LIN {X 0,Y 320.204,Z 957.496,A -85,B 0,C 180,E1 15355.155,E2 15355.155} C_VEL
LIN {X 0,Y 325.919,Z 943.483,A -85,B 0,C 180,E1 15351.712,E2 15351.712} C_VEL
LIN {X 0,Y 332.277,Z 928.194,A -85,B 0,C 180,E1 15348.526,E2 15348.526} C_VEL
LIN {X 0,Y 338.79,Z 912.192,A -85,B 0,C 180,E1 15345.742,E2 15345.742} C_VEL
LIN {X 0,Y 346.075,Z 893.682,A -85,B 0,C 180,E1 15343.041,E2 15343.041} C_VEL
LIN {X 0,Y 352.439,Z 876.534,A -85,B 0,C 180,E1 15340.945,E2 15340.945} C_VEL
LIN {X 0,Y 359.474,Z 856.024,A -85,B 0,C 180,E1 15338.858,E2 15338.858} C_VEL
LIN {X 0,Y 365.817,Z 835.8,A -85,B 0,C 180,E1 15337.159,E2 15337.159} C_VEL
LIN {X 0,Y 371.591,Z 814.628,A -85,B 0,C 180,E1 15335.724,E2 15335.724} C_VEL
LIN {X 0,Y 376.805,Z 792.847,A -85,B 0,C 180,E1 15334.531,E2 15334.531} C_VEL
LIN {X 0,Y 381.083,Z 770.761,A -85,B 0,C 180,E1 15333.6,E2 15333.6} C_VEL
LIN {X 0,Y 384.81,Z 746.357,A -85,B 0,C 180,E1 15332.838,E2 15332.838} C_VEL
LIN {X 0,Y 387.003,Z 723.943,A -85,B 0,C 180,E1 15332.314,E2 15332.314} C_VEL
LIN {X 0,Y 400.127,Z 517.073,A -85,B 0,C 180,E1 15328.257,E2 15328.257} C_VEL
LIN {X 0,Y 400.762,Z 506.979,A -85,B 0,C 180,E1 15328.052,E2 15328.052} C_VEL
LIN {X 0,Y 392.665,Z 493.102,A -85,B 0,C 180,E1 15325.206,E2 15325.206} C_VEL
LIN {X 0,Y 385.414,Z 481.504,A -85,B 0,C 180,E1 15322.297,E2 15322.297} C_VEL
LIN {X 0,Y 380.756,Z 474.893,A -85,B 0,C 180,E1 15320.201,E2 15320.201} C_VEL
LIN {X 0,Y 377.273,Z 470.183,A -85,B 0,C 180,E1 15318.463,E2 15318.463} C_VEL
LIN {X 0,Y 373.457,Z 465.169,A -85,B 0,C 180,E1 15316.326,E2 15316.326} C_VEL
LIN {X 0,Y 370.115,Z 460.624,A -85,B 0,C 180,E1 15314.151,E2 15314.151} C_VEL
LIN {X 0,Y 366.362,Z 456.303,A -85,B 0,C 180,E1 15311.252,E2 15311.252} C_VEL
LIN {X 0,Y 365.344,Z 454.428,A -85,B 0,C 180,E1 15310.246,E2 15310.246} C_VEL
LIN {X 0,Y 362.011,Z 451.144,A -85,B 0,C 180,E1 15306.342,E2 15306.342} C_VEL
LIN {X 0,Y 360.93,Z 448.352,A -85,B 0,C 180,E1 15303.971,E2 15303.971} C_VEL
LIN {X 0,Y 360.463,Z 448.211,A -85,B 0,C 180,E1 15296.66,E2 15296.66} C_VEL
LIN {X 0,Y 361.126,Z 448.613,A -85,B 0,C 180,E1 15294.996,E2 15294.996} C_VEL
LIN {X 0,Y 362.687,Z 452.129,A -85,B 0,C 180,E1 15292.077,E2 15292.077} C_VEL
LIN {X 0,Y 365.646,Z 454.865,A -85,B 0,C 180,E1 15288.884,E2 15288.884} C_VEL
LIN {X 0,Y 368.285,Z 458.822,A -85,B 0,C 180,E1 15286.578,E2 15286.578} C_VEL
LIN {X 0,Y 370.2,Z 460.795,A -85,B 0,C 180,E1 15285.212,E2 15285.212} C_VEL
LIN {X 0,Y 373.571,Z 465.247,A -85,B 0,C 180,E1 15283.038,E2 15283.038} C_VEL
LIN {X 0,Y 378.886,Z 472.366,A -85,B 0,C 180,E1 15280.137,E2 15280.137} C_VEL
LIN {X 0,Y 382.899,Z 477.884,A -85,B 0,C 180,E1 15278.235,E2 15278.235} C_VEL
LIN {X 0,Y 388.744,Z 485.936,A -85,B 0,C 180,E1 15275.78,E2 15275.78} C_VEL
LIN {X 0,Y 397.542,Z 499.019,A -85,B 0,C 180,E1 15272.555,E2 15272.555} C_VEL
LIN {X 0,Y 400.68,Z 504.305,A -85,B 0,C 180,E1 15271.496,E2 15271.496} C_VEL
LIN {X 0,Y 387.414,Z 710.788,A -85,B 0,C 180,E1 15267.448,E2 15267.448} C_VEL
LIN {X 0,Y 385.19,Z 733.04,A -85,B 0,C 180,E1 15266.904,E2 15266.904} C_VEL
LIN {X 0,Y 381.856,Z 755.375,A -85,B 0,C 180,E1 15266.142,E2 15266.142} C_VEL
LIN {X 0,Y 377.948,Z 776.257,A -85,B 0,C 180,E1 15265.218,E2 15265.218} C_VEL
LIN {X 0,Y 373.062,Z 797.329,A -85,B 0,C 180,E1 15264.028,E2 15264.028} C_VEL
LIN {X 0,Y 367.712,Z 817.41,A -85,B 0,C 180,E1 15262.642,E2 15262.642} C_VEL
LIN {X 0,Y 361.615,Z 837.121,A -85,B 0,C 180,E1 15260.974,E2 15260.974} C_VEL
LIN {X 0,Y 355.259,Z 855.944,A -85,B 0,C 180,E1 15259.074,E2 15259.074} C_VEL
LIN {X 0,Y 348.293,Z 874.444,A -85,B 0,C 180,E1 15256.809,E2 15256.809} C_VEL
LIN {X 0,Y 341.213,Z 892.21,A -85,B 0,C 180,E1 15254.213,E2 15254.213} C_VEL
LIN {X 0,Y 334.762,Z 907.539,A -85,B 0,C 180,E1 15251.527,E2 15251.527} C_VEL
LIN {X 0,Y 327.933,Z 923.307,A -85,B 0,C 180,E1 15248.233,E2 15248.233} C_VEL
LIN {X 0,Y 322.331,Z 936.215,A -85,B 0,C 180,E1 15245.015,E2 15245.015} C_VEL
LIN {X 0,Y 316.952,Z 948.748,A -85,B 0,C 180,E1 15241.251,E2 15241.251} C_VEL
LIN {X 0,Y 312.67,Z 959.438,A -85,B 0,C 180,E1 15237.414,E2 15237.414} C_VEL
LIN {X 0,Y 309.22,Z 968.65,A -85,B 0,C 180,E1 15233.319,E2 15233.319} C_VEL
LIN {X 0,Y 306.721,Z 976.512,A -85,B 0,C 180,E1 15229.022,E2 15229.022} C_VEL
LIN {X 0,Y 305.297,Z 981.991,A -85,B 0,C 180,E1 15225.187,E2 15225.187} C_VEL
LIN {X 0,Y 304.432,Z 986.613,A -85,B 0,C 180,E1 15220.98,E2 15220.98} C_VEL
LIN {X 0,Y 304.083,Z 989.403,A -85,B 0,C 180,E1 15217.176,E2 15217.176} C_VEL
LIN {X 0,Y 303.978,Z 991.015,A -85,B 0,C 180,E1 15213.582,E2 15213.582} C_VEL
LIN {X 0,Y 303.96,Z 991.586,A -85,B 0,C 180,E1 15209.623,E2 15209.623} C_VEL
LIN {X 0,Y 303.993,Z 990.851,A -85,B 0,C 180,E1 15205.85,E2 15205.85} C_VEL
LIN {X 0,Y 304.109,Z 989.131,A -85,B 0,C 180,E1 15202.253,E2 15202.253} C_VEL
LIN {X 0,Y 304.564,Z 985.749,A -85,B 0,C 180,E1 15198.045,E2 15198.045} C_VEL
LIN {X 0,Y 305.44,Z 981.375,A -85,B 0,C 180,E1 15194.236,E2 15194.236} C_VEL
LIN {X 0,Y 305.492,Z 981.166,A -85,B 0,C 180,E1 15194.073,E2 15194.073} C_VEL
LIN {X 0,Y 305.002,Z 979.368,A -85,B 0,C 180,E1 15192.66,E2 15192.66} C_VEL
LIN {X 0,Y 300.55,Z 974.185,A -85,B 0,C 180,E1 15188.845,E2 15188.845} C_VEL
LIN {X 0,Y 300.527,Z 972.173,A -85,B 0,C 180,E1 15187.629,E2 15187.629} C_VEL
LIN {X 0,Y 303.768,Z 963.538,A -85,B 0,C 180,E1 15183.41,E2 15183.41} C_VEL
LIN {X 0,Y 307.801,Z 953.96,A -85,B 0,C 180,E1 15179.556,E2 15179.556} C_VEL
LIN {X 0,Y 312.845,Z 942.539,A -85,B 0,C 180,E1 15175.775,E2 15175.775} C_VEL
LIN {X 0,Y 318.733,Z 929.796,A -85,B 0,C 180,E1 15172.234,E2 15172.234} C_VEL
LIN {X 0,Y 325.37,Z 915.155,A -85,B 0,C 180,E1 15168.887,E2 15168.887} C_VEL
LIN {X 0,Y 332.637,Z 898.955,A -85,B 0,C 180,E1 15165.79,E2 15165.79} C_VEL
LIN {X 0,Y 339.295,Z 883.331,A -85,B 0,C 180,E1 15163.298,E2 15163.298} C_VEL
LIN {X 0,Y 346.999,Z 864.093,A -85,B 0,C 180,E1 15160.735,E2 15160.735} C_VEL
LIN {X 0,Y 353.709,Z 845.967,A -85,B 0,C 180,E1 15158.729,E2 15158.729} C_VEL
LIN {X 0,Y 360.218,Z 826.344,A -85,B 0,C 180,E1 15156.935,E2 15156.935} C_VEL
LIN {X 0,Y 366.181,Z 806.306,A -85,B 0,C 180,E1 15155.416,E2 15155.416} C_VEL
LIN {X 0,Y 371.435,Z 785.463,A -85,B 0,C 180,E1 15154.14,E2 15154.14} C_VEL
LIN {X 0,Y 376.179,Z 763.349,A -85,B 0,C 180,E1 15153.053,E2 15153.053} C_VEL
LIN {X 0,Y 379.818,Z 741.232,A -85,B 0,C 180,E1 15152.229,E2 15152.229} C_VEL
LIN {X 0,Y 382.735,Z 717.296,A -85,B 0,C 180,E1 15151.579,E2 15151.579} C_VEL
LIN {X 0,Y 395.368,Z 528.784,A -85,B 0,C 180,E1 15147.863,E2 15147.863} C_VEL
LIN {X 0,Y 396.731,Z 508.619,A -85,B 0,C 180,E1 15147.465,E2 15147.465} C_VEL
LIN {X 0,Y 389.098,Z 496.82,A -85,B 0,C 180,E1 15144.682,E2 15144.682} C_VEL
LIN {X 0,Y 382.445,Z 487.221,A -85,B 0,C 180,E1 15141.914,E2 15141.914} C_VEL
LIN {X 0,Y 378.4,Z 481.609,A -85,B 0,C 180,E1 15140.01,E2 15140.01} C_VEL
LIN {X 0,Y 375.455,Z 477.526,A -85,B 0,C 180,E1 15138.476,E2 15138.476} C_VEL
LIN {X 0,Y 372.006,Z 472.824,A -85,B 0,C 180,E1 15136.473,E2 15136.473} C_VEL
LIN {X 0,Y 368.649,Z 468.169,A -85,B 0,C 180,E1 15134.209,E2 15134.209} C_VEL
LIN {X 0,Y 365.046,Z 463.88,A -85,B 0,C 180,E1 15131.294,E2 15131.294} C_VEL
LIN {X 0,Y 364.061,Z 462.185,A -85,B 0,C 180,E1 15130.284,E2 15130.284} C_VEL
LIN {X 0,Y 360.943,Z 458.912,A -85,B 0,C 180,E1 15126.362,E2 15126.362} C_VEL
LIN {X 0,Y 360.04,Z 456.293,A -85,B 0,C 180,E1 15124.141,E2 15124.141} C_VEL
LIN {X 0,Y 359.977,Z 456.281,A -85,B 0,C 180,E1 15116.497,E2 15116.497} C_VEL
LIN {X 0,Y 362.455,Z 460.975,A -85,B 0,C 180,E1 15111.913,E2 15111.913} C_VEL
LIN {X 0,Y 364.452,Z 462.647,A -85,B 0,C 180,E1 15109.808,E2 15109.808} C_VEL
LIN {X 0,Y 367.084,Z 466.751,A -85,B 0,C 180,E1 15107.415,E2 15107.415} C_VEL
LIN {X 0,Y 368.85,Z 468.542,A -85,B 0,C 180,E1 15106.12,E2 15106.12} C_VEL
LIN {X 0,Y 372.256,Z 473.092,A -85,B 0,C 180,E1 15103.86,E2 15103.86} C_VEL
LIN {X 0,Y 377.256,Z 479.962,A -85,B 0,C 180,E1 15101.055,E2 15101.055} C_VEL
LIN {X 0,Y 381.18,Z 485.5,A -85,B 0,C 180,E1 15099.141,E2 15099.141} C_VEL
LIN {X 0,Y 385.654,Z 492.449,A -85,B 0,C 180,E1 15097.155,E2 15097.155} C_VEL
LIN {X 0,Y 392.548,Z 503.898,A -85,B 0,C 180,E1 15094.423,E2 15094.423} C_VEL
LIN {X 0,Y 396.813,Z 511.775,A -85,B 0,C 180,E1 15092.873,E2 15092.873} C_VEL
LIN {X 0,Y 383.039,Z 721.232,A -85,B 0,C 180,E1 15088.764,E2 15088.764} C_VEL
LIN {X 0,Y 380.765,Z 744.543,A -85,B 0,C 180,E1 15088.226,E2 15088.226} C_VEL
LIN {X 0,Y 377.031,Z 768.994,A -85,B 0,C 180,E1 15087.482,E2 15087.482} C_VEL
LIN {X 0,Y 373.092,Z 788.994,A -85,B 0,C 180,E1 15086.662,E2 15086.662} C_VEL
LIN {X 0,Y 367.684,Z 811.66,A -85,B 0,C 180,E1 15085.474,E2 15085.474} C_VEL
LIN {X 0,Y 362.223,Z 831.325,A -85,B 0,C 180,E1 15084.184,E2 15084.184} C_VEL
LIN {X 0,Y 355.5,Z 852.565,A -85,B 0,C 180,E1 15082.472,E2 15082.472} C_VEL
LIN {X 0,Y 348.764,Z 871.867,A -85,B 0,C 180,E1 15080.582,E2 15080.582} C_VEL
LIN {X 0,Y 341.43,Z 890.989,A -85,B 0,C 180,E1 15078.303,E2 15078.303} C_VEL
LIN {X 0,Y 334.217,Z 908.855,A -85,B 0,C 180,E1 15075.76,E2 15075.76} C_VEL
LIN {X 0,Y 327.211,Z 925.222,A -85,B 0,C 180,E1 15072.949,E2 15072.949} C_VEL
LIN {X 0,Y 320.072,Z 941.638,A -85,B 0,C 180,E1 15069.583,E2 15069.583} C_VEL
LIN {X 0,Y 314.248,Z 955.086,A -85,B 0,C 180,E1 15066.281,E2 15066.281} C_VEL
LIN {X 0,Y 308.813,Z 967.94,A -85,B 0,C 180,E1 15062.508,E2 15062.508} C_VEL
LIN {X 0,Y 304.281,Z 979.499,A -85,B 0,C 180,E1 15058.452,E2 15058.452} C_VEL
LIN {X 0,Y 300.872,Z 989.048,A -85,B 0,C 180,E1 15054.333,E2 15054.333} C_VEL
LIN {X 0,Y 298.43,Z 997.374,A -85,B 0,C 180,E1 15049.981,E2 15049.981} C_VEL
LIN {X 0,Y 296.983,Z 1003.564,A -85,B 0,C 180,E1 15045.824,E2 15045.824} C_VEL
LIN {X 0,Y 296.221,Z 1008.587,A -85,B 0,C 180,E1 15041.486,E2 15041.486} C_VEL
LIN {X 0,Y 295.976,Z 1011.635,A -85,B 0,C 180,E1 15037.57,E2 15037.57} C_VEL
LIN {X 0,Y 295.96,Z 1013.344,A -85,B 0,C 180,E1 15034.068,E2 15034.068} C_VEL
LIN {X 0,Y 295.977,Z 1014.117,A -85,B 0,C 180,E1 15030.001,E2 15030.001} C_VEL
LIN {X 0,Y 295.959,Z 1013.342,A -85,B 0,C 180,E1 15025.933,E2 15025.933} C_VEL
LIN {X 0,Y 295.977,Z 1011.631,A -85,B 0,C 180,E1 15022.431,E2 15022.431} C_VEL
LIN {X 0,Y 296.241,Z 1008.39,A -85,B 0,C 180,E1 15018.318,E2 15018.318} C_VEL
LIN {X 0,Y 296.982,Z 1003.558,A -85,B 0,C 180,E1 15014.177,E2 15014.177} C_VEL
LIN {X 0,Y 298.428,Z 997.364,A -85,B 0,C 180,E1 15010.02,E2 15010.02} C_VEL
LIN {X 0,Y 300.874,Z 989.034,A -85,B 0,C 180,E1 15005.668,E2 15005.668} C_VEL
LIN {X 0,Y 304.278,Z 979.484,A -85,B 0,C 180,E1 15001.549,E2 15001.549} C_VEL
LIN {X 0,Y 308.808,Z 967.92,A -85,B 0,C 180,E1 14997.493,E2 14997.493} C_VEL
LIN {X 0,Y 314.542,Z 954.339,A -85,B 0,C 180,E1 14993.533,E2 14993.533} C_VEL
LIN {X 0,Y 320.416,Z 940.813,A -85,B 0,C 180,E1 14990.237,E2 14990.237} C_VEL
LIN {X 0,Y 327.404,Z 924.699,A -85,B 0,C 180,E1 14986.964,E2 14986.964} C_VEL
LIN {X 0,Y 334.431,Z 908.269,A -85,B 0,C 180,E1 14984.155,E2 14984.155} C_VEL
LIN {X 0,Y 341.586,Z 890.474,A -85,B 0,C 180,E1 14981.64,E2 14981.64} C_VEL
LIN {X 0,Y 349.009,Z 871.012,A -85,B 0,C 180,E1 14979.339,E2 14979.339} C_VEL
LIN {X 0,Y 355.484,Z 852.438,A -85,B 0,C 180,E1 14977.526,E2 14977.526} C_VEL
LIN {X 0,Y 362.323,Z 830.765,A -85,B 0,C 180,E1 14975.785,E2 14975.785} C_VEL
LIN {X 0,Y 367.666,Z 811.477,A -85,B 0,C 180,E1 14974.523,E2 14974.523} C_VEL
LIN {X 0,Y 372.9,Z 789.56,A -85,B 0,C 180,E1 14973.371,E2 14973.371} C_VEL
LIN {X 0,Y 376.938,Z 769.089,A -85,B 0,C 180,E1 14972.529,E2 14972.529} C_VEL
LIN {X 0,Y 380.682,Z 744.574,A -85,B 0,C 180,E1 14971.782,E2 14971.782} C_VEL
LIN {X 0,Y 382.974,Z 721.037,A -85,B 0,C 180,E1 14971.24,E2 14971.24} C_VEL
LIN {X 0,Y 396.738,Z 511.466,A -85,B 0,C 180,E1 14967.129,E2 14967.129} C_VEL
LIN {X 0,Y 389.576,Z 498.912,A -85,B 0,C 180,E1 14964.487,E2 14964.487} C_VEL
LIN {X 0,Y 382.313,Z 487.129,A -85,B 0,C 180,E1 14961.433,E2 14961.433} C_VEL
LIN {X 0,Y 378.126,Z 481.293,A -85,B 0,C 180,E1 14959.461,E2 14959.461} C_VEL
LIN {X 0,Y 375.458,Z 477.57,A -85,B 0,C 180,E1 14958.074,E2 14958.074} C_VEL
LIN {X 0,Y 371.857,Z 472.733,A -85,B 0,C 180,E1 14955.998,E2 14955.998} C_VEL
LIN {X 0,Y 368.172,Z 467.718,A -85,B 0,C 180,E1 14953.506,E2 14953.506} C_VEL
LIN {X 0,Y 365.12,Z 464.139,A -85,B 0,C 180,E1 14951.051,E2 14951.051} C_VEL
LIN {X 0,Y 364.041,Z 462.222,A -85,B 0,C 180,E1 14949.964,E2 14949.964} C_VEL
LIN {X 0,Y 360.758,Z 458.669,A -85,B 0,C 180,E1 14945.885,E2 14945.885} C_VEL
LIN {X 0,Y 359.886,Z 456.277,A -85,B 0,C 180,E1 14943.823,E2 14943.823} C_VEL
LIN {X 0,Y 359.49,Z 456.153,A -85,B 0,C 180,E1 14936.651,E2 14936.651} C_VEL
LIN {X 0,Y 360.073,Z 456.551,A -85,B 0,C 180,E1 14935.141,E2 14935.141} C_VEL
LIN {X 0,Y 361.71,Z 460.167,A -85,B 0,C 180,E1 14932.055,E2 14932.055} C_VEL
LIN {X 0,Y 364.345,Z 462.578,A -85,B 0,C 180,E1 14929.165,E2 14929.165} C_VEL
LIN {X 0,Y 367.015,Z 466.623,A -85,B 0,C 180,E1 14926.771,E2 14926.771} C_VEL
LIN {X 0,Y 368.784,Z 468.533,A -85,B 0,C 180,E1 14925.476,E2 14925.476} C_VEL
LIN {X 0,Y 372.353,Z 473.176,A -85,B 0,C 180,E1 14923.141,E2 14923.141} C_VEL
LIN {X 0,Y 377.32,Z 480.16,A -85,B 0,C 180,E1 14920.374,E2 14920.374} C_VEL
LIN {X 0,Y 381.277,Z 485.71,A -85,B 0,C 180,E1 14918.461,E2 14918.461} C_VEL
LIN {X 0,Y 386.702,Z 493.369,A -85,B 0,C 180,E1 14916.131,E2 14916.131} C_VEL
LIN {X 0,Y 394.978,Z 505.909,A -85,B 0,C 180,E1 14913.015,E2 14913.015} C_VEL
LIN {X 0,Y 396.636,Z 508.825,A -85,B 0,C 180,E1 14912.429,E2 14912.429} C_VEL
LIN {X 0,Y 382.999,Z 713.139,A -85,B 0,C 180,E1 14908.413,E2 14908.413} C_VEL
LIN {X 0,Y 380.495,Z 736.296,A -85,B 0,C 180,E1 14907.828,E2 14907.828} C_VEL
LIN {X 0,Y 377.14,Z 757.433,A -85,B 0,C 180,E1 14907.084,E2 14907.084} C_VEL
LIN {X 0,Y 372.84,Z 779.225,A -85,B 0,C 180,E1 14906.096,E2 14906.096} C_VEL
LIN {X 0,Y 368.092,Z 798.762,A -85,B 0,C 180,E1 14904.972,E2 14904.972} C_VEL
LIN {X 0,Y 362.377,Z 819.346,A -85,B 0,C 180,E1 14903.533,E2 14903.533} C_VEL
LIN {X 0,Y 356.288,Z 838.235,A -85,B 0,C 180,E1 14901.913,E2 14901.913} C_VEL
LIN {X 0,Y 349.442,Z 857.624,A -85,B 0,C 180,E1 14899.925,E2 14899.925} C_VEL
LIN {X 0,Y 342.507,Z 875.356,A -85,B 0,C 180,E1 14897.726,E2 14897.726} C_VEL
LIN {X 0,Y 334.93,Z 893.521,A -85,B 0,C 180,E1 14895.025,E2 14895.025} C_VEL
LIN {X 0,Y 328.24,Z 908.763,A -85,B 0,C 180,E1 14892.307,E2 14892.307} C_VEL
LIN {X 0,Y 321.133,Z 924.376,A -85,B 0,C 180,E1 14888.966,E2 14888.966} C_VEL
LIN {X 0,Y 314.996,Z 937.894,A -85,B 0,C 180,E1 14885.507,E2 14885.507} C_VEL
LIN {X 0,Y 309.541,Z 949.889,A -85,B 0,C 180,E1 14881.765,E2 14881.765} C_VEL
LIN {X 0,Y 304.921,Z 960.735,A -85,B 0,C 180,E1 14877.705,E2 14877.705} C_VEL
LIN {X 0,Y 301.465,Z 969.527,A -85,B 0,C 180,E1 14873.657,E2 14873.657} C_VEL
LIN {X 0,Y 298.79,Z 977.408,A -85,B 0,C 180,E1 14869.141,E2 14869.141} C_VEL
LIN {X 0,Y 297.313,Z 982.841,A -85,B 0,C 180,E1 14865.164,E2 14865.164} C_VEL
LIN {X 0,Y 296.401,Z 987.378,A -85,B 0,C 180,E1 14860.69,E2 14860.69} C_VEL
LIN {X 0,Y 296.088,Z 989.923,A -85,B 0,C 180,E1 14856.981,E2 14856.981} C_VEL
LIN {X 0,Y 295.978,Z 991.578,A -85,B 0,C 180,E1 14852.904,E2 14852.904} C_VEL
LIN {X 0,Y 295.97,Z 991.797,A -85,B 0,C 180,E1 14848.838,E2 14848.838} C_VEL
LIN {X 0,Y 296.012,Z 990.956,A -85,B 0,C 180,E1 14845.156,E2 14845.156} C_VEL
LIN {X 0,Y 296.246,Z 988.685,A -85,B 0,C 180,E1 14840.873,E2 14840.873} C_VEL
LIN {X 0,Y 296.826,Z 985.074,A -85,B 0,C 180,E1 14836.759,E2 14836.759} C_VEL
LIN {X 0,Y 298.103,Z 979.901,A -85,B 0,C 180,E1 14832.432,E2 14832.432} C_VEL
LIN {X 0,Y 300.117,Z 973.342,A -85,B 0,C 180,E1 14828.299,E2 14828.299} C_VEL
LIN {X 0,Y 300.527,Z 972.173,A -85,B 0,C 180,E1 14827.629,E2 14827.629} C_VEL
LIN {X 0,Y 300.487,Z 969.761,A -85,B 0,C 180,E1 14826.222,E2 14826.222} C_VEL
LIN {X 0,Y 297.448,Z 963.001,A -85,B 0,C 180,E1 14822.402,E2 14822.402} C_VEL
LIN {X 0,Y 297.9,Z 960.498,A -85,B 0,C 180,E1 14821.214,E2 14821.214} C_VEL
LIN {X 0,Y 302.703,Z 949.892,A -85,B 0,C 180,E1 14817.204,E2 14817.204} C_VEL
LIN {X 0,Y 308.491,Z 937.836,A -85,B 0,C 180,E1 14813.394,E2 14813.394} C_VEL
LIN {X 0,Y 314.996,Z 924.269,A -85,B 0,C 180,E1 14809.887,E2 14809.887} C_VEL
LIN {X 0,Y 322.462,Z 908.563,A -85,B 0,C 180,E1 14806.506,E2 14806.506} C_VEL
LIN {X 0,Y 329.485,Z 893.265,A -85,B 0,C 180,E1 14803.767,E2 14803.767} C_VEL
LIN {X 0,Y 337.154,Z 875.582,A -85,B 0,C 180,E1 14801.133,E2 14801.133} C_VEL
LIN {X 0,Y 344.109,Z 858.451,A -85,B 0,C 180,E1 14798.997,E2 14798.997} C_VEL
LIN {X 0,Y 351.174,Z 839.22,A -85,B 0,C 180,E1 14797.008,E2 14797.008} C_VEL
LIN {X 0,Y 357.477,Z 820.322,A -85,B 0,C 180,E1 14795.379,E2 14795.379} C_VEL
LIN {X 0,Y 363.453,Z 799.617,A -85,B 0,C 180,E1 14793.923,E2 14793.923} C_VEL
LIN {X 0,Y 368.536,Z 779.372,A -85,B 0,C 180,E1 14792.759,E2 14792.759} C_VEL
LIN {X 0,Y 372.971,Z 757.496,A -85,B 0,C 180,E1 14791.773,E2 14791.773} C_VEL
LIN {X 0,Y 376.474,Z 736.015,A -85,B 0,C 180,E1 14791.024,E2 14791.024} C_VEL
LIN {X 0,Y 379.006,Z 712.92,A -85,B 0,C 180,E1 14790.447,E2 14790.447} C_VEL
LIN {X 0,Y 392.799,Z 513.344,A -85,B 0,C 180,E1 14786.52,E2 14786.52} C_VEL
LIN {X 0,Y 386.251,Z 503.102,A -85,B 0,C 180,E1 14784.021,E2 14784.021} C_VEL
LIN {X 0,Y 380.27,Z 494.271,A -85,B 0,C 180,E1 14781.437,E2 14781.437} C_VEL
LIN {X 0,Y 376.118,Z 488.381,A -85,B 0,C 180,E1 14779.408,E2 14779.408} C_VEL
LIN {X 0,Y 373.531,Z 484.746,A -85,B 0,C 180,E1 14778.009,E2 14778.009} C_VEL
LIN {X 0,Y 370.422,Z 480.39,A -85,B 0,C 180,E1 14776.142,E2 14776.142} C_VEL
LIN {X 0,Y 366.736,Z 475.317,A -85,B 0,C 180,E1 14773.561,E2 14773.561} C_VEL
LIN {X 0,Y 363.666,Z 471.428,A -85,B 0,C 180,E1 14770.936,E2 14770.936} C_VEL
LIN {X 0,Y 362.935,Z 470.068,A -85,B 0,C 180,E1 14770.156,E2 14770.156} C_VEL
LIN {X 0,Y 359.875,Z 466.798,A -85,B 0,C 180,E1 14766.221,E2 14766.221} C_VEL
LIN {X 0,Y 359.003,Z 464.22,A -85,B 0,C 180,E1 14763.993,E2 14763.993} C_VEL
LIN {X 0,Y 359.035,Z 464.233,A -85,B 0,C 180,E1 14756.408,E2 14756.408} C_VEL
LIN {X 0,Y 360.99,Z 468.49,A -85,B 0,C 180,E1 14752.511,E2 14752.511} C_VEL
LIN {X 0,Y 363.232,Z 470.516,A -85,B 0,C 180,E1 14750.014,E2 14750.014} C_VEL
LIN {X 0,Y 365.916,Z 474.648,A -85,B 0,C 180,E1 14747.534,E2 14747.534} C_VEL
LIN {X 0,Y 367.445,Z 476.272,A -85,B 0,C 180,E1 14746.387,E2 14746.387} C_VEL
LIN {X 0,Y 371.621,Z 482.099,A -85,B 0,C 180,E1 14743.591,E2 14743.591} C_VEL
LIN {X 0,Y 375.472,Z 487.399,A -85,B 0,C 180,E1 14741.417,E2 14741.417} C_VEL
LIN {X 0,Y 379.643,Z 493.425,A -85,B 0,C 180,E1 14739.335,E2 14739.335} C_VEL
LIN {X 0,Y 384.555,Z 501.294,A -85,B 0,C 180,E1 14737.126,E2 14737.126} C_VEL
LIN {X 0,Y 391.313,Z 513.083,A -85,B 0,C 180,E1 14734.417,E2 14734.417} C_VEL
LIN {X 0,Y 392.867,Z 516.259,A -85,B 0,C 180,E1 14733.825,E2 14733.825} C_VEL
LIN {X 0,Y 378.717,Z 723.42,A -85,B 0,C 180,E1 14729.751,E2 14729.751} C_VEL
LIN {X 0,Y 376.409,Z 745.722,A -85,B 0,C 180,E1 14729.23,E2 14729.23} C_VEL
LIN {X 0,Y 372.491,Z 770.088,A -85,B 0,C 180,E1 14728.477,E2 14728.477} C_VEL
LIN {X 0,Y 368.209,Z 791.004,A -85,B 0,C 180,E1 14727.61,E2 14727.61} C_VEL
LIN {X 0,Y 362.824,Z 812.499,A -85,B 0,C 180,E1 14726.463,E2 14726.463} C_VEL
LIN {X 0,Y 357.028,Z 832.644,A -85,B 0,C 180,E1 14725.131,E2 14725.131} C_VEL
LIN {X 0,Y 350.215,Z 853.249,A -85,B 0,C 180,E1 14723.446,E2 14723.446} C_VEL
LIN {X 0,Y 343.071,Z 872.959,A -85,B 0,C 180,E1 14721.497,E2 14721.497} C_VEL
LIN {X 0,Y 335.466,Z 891.912,A -85,B 0,C 180,E1 14719.198,E2 14719.198} C_VEL
LIN {X 0,Y 327.527,Z 910.601,A -85,B 0,C 180,E1 14716.465,E2 14716.465} C_VEL
LIN {X 0,Y 320.518,Z 926.321,A -85,B 0,C 180,E1 14713.701,E2 14713.701} C_VEL
LIN {X 0,Y 313.287,Z 942.11,A -85,B 0,C 180,E1 14710.377,E2 14710.377} C_VEL
LIN {X 0,Y 306.899,Z 956.201,A -85,B 0,C 180,E1 14706.827,E2 14706.827} C_VEL
LIN {X 0,Y 301.255,Z 968.799,A -85,B 0,C 180,E1 14702.974,E2 14702.974} C_VEL
LIN {X 0,Y 296.547,Z 980.162,A -85,B 0,C 180,E1 14698.823,E2 14698.823} C_VEL
LIN {X 0,Y 293.009,Z 989.569,A -85,B 0,C 180,E1 14694.599,E2 14694.599} C_VEL
LIN {X 0,Y 290.382,Z 998.004,A -85,B 0,C 180,E1 14689.929,E2 14689.929} C_VEL
LIN {X 0,Y 288.984,Z 1003.783,A -85,B 0,C 180,E1 14685.861,E2 14685.861} C_VEL
LIN {X 0,Y 288.213,Z 1008.616,A -85,B 0,C 180,E1 14681.404,E2 14681.404} C_VEL
LIN {X 0,Y 287.978,Z 1011.451,A -85,B 0,C 180,E1 14677.581,E2 14677.581} C_VEL
LIN {X 0,Y 287.962,Z 1013.114,A -85,B 0,C 180,E1 14673.982,E2 14673.982} C_VEL
LIN {X 0,Y 287.982,Z 1013.817,A -85,B 0,C 180,E1 14670.001,E2 14670.001} C_VEL
LIN {X 0,Y 287.962,Z 1013.112,A -85,B 0,C 180,E1 14666.019,E2 14666.019} C_VEL
LIN {X 0,Y 287.98,Z 1011.447,A -85,B 0,C 180,E1 14662.42,E2 14662.42} C_VEL
LIN {X 0,Y 288.232,Z 1008.444,A -85,B 0,C 180,E1 14658.395,E2 14658.395} C_VEL
LIN {X 0,Y 289.037,Z 1003.512,A -85,B 0,C 180,E1 14653.937,E2 14653.937} C_VEL
LIN {X 0,Y 290.564,Z 997.366,A -85,B 0,C 180,E1 14649.665,E2 14649.665} C_VEL
LIN {X 0,Y 293.154,Z 989.137,A -85,B 0,C 180,E1 14645.2,E2 14645.2} C_VEL
LIN {X 0,Y 296.743,Z 979.675,A -85,B 0,C 180,E1 14640.979,E2 14640.979} C_VEL
LIN {X 0,Y 301.501,Z 968.19,A -85,B 0,C 180,E1 14636.831,E2 14636.831} C_VEL
LIN {X 0,Y 307.202,Z 955.451,A -85,B 0,C 180,E1 14632.983,E2 14632.983} C_VEL
LIN {X 0,Y 313.279,Z 942.065,A -85,B 0,C 180,E1 14629.623,E2 14629.623} C_VEL
LIN {X 0,Y 320.926,Z 925.323,A -85,B 0,C 180,E1 14626.123,E2 14626.123} C_VEL
LIN {X 0,Y 327.976,Z 909.505,A -85,B 0,C 180,E1 14623.365,E2 14623.365} C_VEL
LIN {X 0,Y 335.452,Z 891.82,A -85,B 0,C 180,E1 14620.801,E2 14620.801} C_VEL
LIN {X 0,Y 343.031,Z 872.905,A -85,B 0,C 180,E1 14618.508,E2 14618.508} C_VEL
LIN {X 0,Y 350.166,Z 853.202,A -85,B 0,C 180,E1 14616.559,E2 14616.559} C_VEL
LIN {X 0,Y 357.01,Z 832.477,A -85,B 0,C 180,E1 14614.866,E2 14614.866} C_VEL
LIN {X 0,Y 362.806,Z 812.303,A -85,B 0,C 180,E1 14613.534,E2 14613.534} C_VEL
LIN {X 0,Y 368.397,Z 789.77,A -85,B 0,C 180,E1 14612.344,E2 14612.344} C_VEL
LIN {X 0,Y 372.533,Z 769.458,A -85,B 0,C 180,E1 14611.508,E2 14611.508} C_VEL
LIN {X 0,Y 376.444,Z 744.746,A -85,B 0,C 180,E1 14610.753,E2 14610.753} C_VEL
LIN {X 0,Y 378.77,Z 721.795,A -85,B 0,C 180,E1 14610.222,E2 14610.222} C_VEL
LIN {X 0,Y 392.789,Z 515.926,A -85,B 0,C 180,E1 14606.176,E2 14606.176} C_VEL
LIN {X 0,Y 386.71,Z 505.109,A -85,B 0,C 180,E1 14603.828,E2 14603.828} C_VEL
LIN {X 0,Y 380.142,Z 494.184,A -85,B 0,C 180,E1 14600.959,E2 14600.959} C_VEL
LIN {X 0,Y 376.056,Z 488.351,A -85,B 0,C 180,E1 14598.967,E2 14598.967} C_VEL
LIN {X 0,Y 373.525,Z 484.794,A -85,B 0,C 180,E1 14597.606,E2 14597.606} C_VEL
LIN {X 0,Y 370.148,Z 480.165,A -85,B 0,C 180,E1 14595.591,E2 14595.591} C_VEL
LIN {X 0,Y 366.778,Z 475.433,A -85,B 0,C 180,E1 14593.237,E2 14593.237} C_VEL
LIN {X 0,Y 363.727,Z 471.685,A -85,B 0,C 180,E1 14590.693,E2 14590.693} C_VEL
LIN {X 0,Y 362.748,Z 470.008,A -85,B 0,C 180,E1 14589.679,E2 14589.679} C_VEL
LIN {X 0,Y 359.688,Z 466.56,A -85,B 0,C 180,E1 14585.743,E2 14585.743} C_VEL
LIN {X 0,Y 358.845,Z 464.199,A -85,B 0,C 180,E1 14583.674,E2 14583.674} C_VEL
LIN {X 0,Y 358.569,Z 464.114,A -85,B 0,C 180,E1 14576.483,E2 14576.483} C_VEL
LIN {X 0,Y 359.025,Z 464.483,A -85,B 0,C 180,E1 14575.287,E2 14575.287} C_VEL
LIN {X 0,Y 360.733,Z 468.202,A -85,B 0,C 180,E1 14572.034,E2 14572.034} C_VEL
LIN {X 0,Y 363.124,Z 470.446,A -85,B 0,C 180,E1 14569.369,E2 14569.369} C_VEL
LIN {X 0,Y 365.847,Z 474.526,A -85,B 0,C 180,E1 14566.889,E2 14566.889} C_VEL
LIN {X 0,Y 367.377,Z 476.266,A -85,B 0,C 180,E1 14565.741,E2 14565.741} C_VEL
LIN {X 0,Y 371.472,Z 481.894,A -85,B 0,C 180,E1 14563.02,E2 14563.02} C_VEL
LIN {X 0,Y 375.552,Z 487.629,A -85,B 0,C 180,E1 14560.723,E2 14560.723} C_VEL
LIN {X 0,Y 379.433,Z 493.191,A -85,B 0,C 180,E1 14558.797,E2 14558.797} C_VEL
LIN {X 0,Y 384.759,Z 500.929,A -85,B 0,C 180,E1 14556.45,E2 14556.45} C_VEL
LIN {X 0,Y 392.441,Z 512.8,A -85,B 0,C 180,E1 14553.48,E2 14553.48} C_VEL
LIN {X 0,Y 392.676,Z 513.682,A -85,B 0,C 180,E1 14553.375,E2 14553.375} C_VEL
LIN {X 0,Y 378.753,Z 714.85,A -85,B 0,C 180,E1 14549.414,E2 14549.414} C_VEL
LIN {X 0,Y 375.922,Z 738.973,A -85,B 0,C 180,E1 14548.786,E2 14548.786} C_VEL
LIN {X 0,Y 372.592,Z 759.14,A -85,B 0,C 180,E1 14548.063,E2 14548.063} C_VEL
LIN {X 0,Y 367.773,Z 782.164,A -85,B 0,C 180,E1 14546.994,E2 14546.994} C_VEL
LIN {X 0,Y 362.928,Z 801.316,A -85,B 0,C 180,E1 14545.87,E2 14545.87} C_VEL
LIN {X 0,Y 356.482,Z 823.135,A -85,B 0,C 180,E1 14544.294,E2 14544.294} C_VEL
LIN {X 0,Y 350.505,Z 840.954,A -85,B 0,C 180,E1 14542.729,E2 14542.729} C_VEL
LIN {X 0,Y 342.937,Z 861.188,A -85,B 0,C 180,E1 14540.582,E2 14540.582} C_VEL
LIN {X 0,Y 335.824,Z 878.672,A -85,B 0,C 180,E1 14538.35,E2 14538.35} C_VEL
LIN {X 0,Y 328.264,Z 895.831,A -85,B 0,C 180,E1 14535.7,E2 14535.7} C_VEL
LIN {X 0,Y 320.968,Z 911.769,A -85,B 0,C 180,E1 14532.767,E2 14532.767} C_VEL
LIN {X 0,Y 314.025,Z 926.202,A -85,B 0,C 180,E1 14529.548,E2 14529.548} C_VEL
LIN {X 0,Y 307.358,Z 940.08,A -85,B 0,C 180,E1 14525.837,E2 14525.837} C_VEL
LIN {X 0,Y 302.022,Z 951.322,A -85,B 0,C 180,E1 14522.204,E2 14522.204} C_VEL
LIN {X 0,Y 297.058,Z 962.3,A -85,B 0,C 180,E1 14517.891,E2 14517.891} C_VEL
LIN {X 0,Y 293.377,Z 971.335,A -85,B 0,C 180,E1 14513.54,E2 14513.54} C_VEL
LIN {X 0,Y 290.766,Z 978.597,A -85,B 0,C 180,E1 14509.064,E2 14509.064} C_VEL
LIN {X 0,Y 289.194,Z 984.288,A -85,B 0,C 180,E1 14504.617,E2 14504.617} C_VEL
LIN {X 0,Y 288.376,Z 988.142,A -85,B 0,C 180,E1 14500.385,E2 14500.385} C_VEL
LIN {X 0,Y 288.086,Z 990.553,A -85,B 0,C 180,E1 14496.575,E2 14496.575} C_VEL
LIN {X 0,Y 287.988,Z 991.977,A -85,B 0,C 180,E1 14492.188,E2 14492.188} C_VEL
LIN {X 0,Y 287.986,Z 992.053,A -85,B 0,C 180,E1 14488.408,E2 14488.408} C_VEL
LIN {X 0,Y 288.052,Z 990.997,A -85,B 0,C 180,E1 14484.223,E2 14484.223} C_VEL
LIN {X 0,Y 288.335,Z 988.519,A -85,B 0,C 180,E1 14480.008,E2 14480.008} C_VEL
LIN {X 0,Y 289.02,Z 984.98,A -85,B 0,C 180,E1 14475.987,E2 14475.987} C_VEL
LIN {X 0,Y 290.553,Z 979.325,A -85,B 0,C 180,E1 14471.337,E2 14471.337} C_VEL
LIN {X 0,Y 292.784,Z 972.844,A -85,B 0,C 180,E1 14467.229,E2 14467.229} C_VEL
LIN {X 0,Y 296.398,Z 963.847,A -85,B 0,C 180,E1 14462.695,E2 14462.695} C_VEL
LIN {X 0,Y 297.9,Z 960.498,A -85,B 0,C 180,E1 14461.214,E2 14461.214} C_VEL
LIN {X 0,Y 298.429,Z 957.538,A -85,B 0,C 180,E1 14459.838,E2 14459.838} C_VEL
LIN {X 0,Y 296.92,Z 949.863,A -85,B 0,C 180,E1 14456.262,E2 14456.262} C_VEL
LIN {X 0,Y 297.809,Z 946.22,A -85,B 0,C 180,E1 14454.951,E2 14454.951} C_VEL
LIN {X 0,Y 304.287,Z 933.333,A -85,B 0,C 180,E1 14451.131,E2 14451.131} C_VEL
LIN {X 0,Y 311.89,Z 918.262,A -85,B 0,C 180,E1 14447.441,E2 14447.441} C_VEL
LIN {X 0,Y 318.761,Z 904.309,A -85,B 0,C 180,E1 14444.606,E2 14444.606} C_VEL
LIN {X 0,Y 326.778,Z 887.225,A -85,B 0,C 180,E1 14441.712,E2 14441.712} C_VEL
LIN {X 0,Y 334.049,Z 870.784,A -85,B 0,C 180,E1 14439.387,E2 14439.387} C_VEL
LIN {X 0,Y 341.785,Z 851.659,A -85,B 0,C 180,E1 14437.147,E2 14437.147} C_VEL
LIN {X 0,Y 348.964,Z 832.276,A -85,B 0,C 180,E1 14435.264,E2 14435.264} C_VEL
LIN {X 0,Y 355.609,Z 811.594,A -85,B 0,C 180,E1 14433.635,E2 14433.635} C_VEL
LIN {X 0,Y 361.716,Z 789.836,A -85,B 0,C 180,E1 14432.242,E2 14432.242} C_VEL
LIN {X 0,Y 366.608,Z 768.776,A -85,B 0,C 180,E1 14431.171,E2 14431.171} C_VEL
LIN {X 0,Y 371.055,Z 744.748,A -85,B 0,C 180,E1 14430.233,E2 14430.233} C_VEL
LIN {X 0,Y 374.204,Z 721.949,A -85,B 0,C 180,E1 14429.584,E2 14429.584} C_VEL
LIN {X 0,Y 377.476,Z 679.365,A -85,B 0,C 180,E1 14428.714,E2 14428.714} C_VEL
LIN {X 0,Y 388.926,Z 517.946,A -85,B 0,C 180,E1 14425.535,E2 14425.535} C_VEL
LIN {X 0,Y 381.576,Z 506.394,A -85,B 0,C 180,E1 14422.534,E2 14422.534} C_VEL
LIN {X 0,Y 375.273,Z 497.097,A -85,B 0,C 180,E1 14419.535,E2 14419.535} C_VEL
LIN {X 0,Y 371.763,Z 492.124,A -85,B 0,C 180,E1 14417.612,E2 14417.612} C_VEL
LIN {X 0,Y 368.774,Z 487.869,A -85,B 0,C 180,E1 14415.76,E2 14415.76} C_VEL
LIN {X 0,Y 365.359,Z 483.026,A -85,B 0,C 180,E1 14413.29,E2 14413.29} C_VEL
LIN {X 0,Y 362.299,Z 478.976,A -85,B 0,C 180,E1 14410.575,E2 14410.575} C_VEL
LIN {X 0,Y 361.654,Z 477.859,A -85,B 0,C 180,E1 14409.87,E2 14409.87} C_VEL
LIN {X 0,Y 358.654,Z 474.338,A -85,B 0,C 180,E1 14405.76,E2 14405.76} C_VEL
LIN {X 0,Y 357.967,Z 472.147,A -85,B 0,C 180,E1 14403.844,E2 14403.844} C_VEL
LIN {X 0,Y 358.014,Z 472.163,A -85,B 0,C 180,E1 14396.518,E2 14396.518} C_VEL
LIN {X 0,Y 359.891,Z 476.36,A -85,B 0,C 180,E1 14392.658,E2 14392.658} C_VEL
LIN {X 0,Y 362.018,Z 478.375,A -85,B 0,C 180,E1 14390.221,E2 14390.221} C_VEL
LIN {X 0,Y 364.75,Z 482.543,A -85,B 0,C 180,E1 14387.654,E2 14387.654} C_VEL
LIN {X 0,Y 366.048,Z 483.999,A -85,B 0,C 180,E1 14386.656,E2 14386.656} C_VEL
LIN {X 0,Y 370.021,Z 489.652,A -85,B 0,C 180,E1 14383.921,E2 14383.921} C_VEL
LIN {X 0,Y 373.81,Z 495.003,A -85,B 0,C 180,E1 14381.723,E2 14381.723} C_VEL
LIN {X 0,Y 378.342,Z 501.644,A -85,B 0,C 180,E1 14379.422,E2 14379.422} C_VEL
LIN {X 0,Y 385.189,Z 513.347,A -85,B 0,C 180,E1 14376.357,E2 14376.357} C_VEL
LIN {X 0,Y 389.047,Z 520.537,A -85,B 0,C 180,E1 14374.8,E2 14374.8} C_VEL
LIN {X 0,Y 374.549,Z 725.174,A -85,B 0,C 180,E1 14370.77,E2 14370.77} C_VEL
LIN {X 0,Y 372.026,Z 748.04,A -85,B 0,C 180,E1 14370.227,E2 14370.227} C_VEL
LIN {X 0,Y 368.059,Z 771.218,A -85,B 0,C 180,E1 14369.495,E2 14369.495} C_VEL
LIN {X 0,Y 363.445,Z 792.91,A -85,B 0,C 180,E1 14368.586,E2 14368.586} C_VEL
LIN {X 0,Y 357.864,Z 814.081,A -85,B 0,C 180,E1 14367.434,E2 14367.434} C_VEL
LIN {X 0,Y 351.495,Z 835.238,A -85,B 0,C 180,E1 14366.007,E2 14366.007} C_VEL
LIN {X 0,Y 344.563,Z 855.232,A -85,B 0,C 180,E1 14364.333,E2 14364.333} C_VEL
LIN {X 0,Y 336.566,Z 876.091,A -85,B 0,C 180,E1 14362.199,E2 14362.199} C_VEL
LIN {X 0,Y 329.072,Z 894.066,A -85,B 0,C 180,E1 14359.96,E2 14359.96} C_VEL
LIN {X 0,Y 320.97,Z 912.174,A -85,B 0,C 180,E1 14357.228,E2 14357.228} C_VEL
LIN {X 0,Y 313.452,Z 928.358,A -85,B 0,C 180,E1 14354.307,E2 14354.307} C_VEL
LIN {X 0,Y 306.187,Z 943.366,A -85,B 0,C 180,E1 14351.018,E2 14351.018} C_VEL
LIN {X 0,Y 299.571,Z 957.233,A -85,B 0,C 180,E1 14347.401,E2 14347.401} C_VEL
LIN {X 0,Y 293.767,Z 969.547,A -85,B 0,C 180,E1 14343.502,E2 14343.502} C_VEL
LIN {X 0,Y 288.622,Z 981.262,A -85,B 0,C 180,E1 14339.009,E2 14339.009} C_VEL
LIN {X 0,Y 285.022,Z 990.467,A -85,B 0,C 180,E1 14334.693,E2 14334.693} C_VEL
LIN {X 0,Y 282.425,Z 998.32,A -85,B 0,C 180,E1 14330.083,E2 14330.083} C_VEL
LIN {X 0,Y 280.93,Z 1004.264,A -85,B 0,C 180,E1 14325.692,E2 14325.692} C_VEL
LIN {X 0,Y 280.182,Z 1008.833,A -85,B 0,C 180,E1 14321.081,E2 14321.081} C_VEL
LIN {X 0,Y 279.971,Z 1011.385,A -85,B 0,C 180,E1 14317.386,E2 14317.386} C_VEL
LIN {X 0,Y 279.958,Z 1013.025,A -85,B 0,C 180,E1 14313.481,E2 14313.481} C_VEL
LIN {X 0,Y 279.971,Z 1013.454,A -85,B 0,C 180,E1 14309.387,E2 14309.387} C_VEL
LIN {X 0,Y 279.966,Z 1012.67,A -85,B 0,C 180,E1 14305.495,E2 14305.495} C_VEL
LIN {X 0,Y 280.034,Z 1010.789,A -85,B 0,C 180,E1 14301.584,E2 14301.584} C_VEL
LIN {X 0,Y 280.447,Z 1006.923,A -85,B 0,C 180,E1 14296.812,E2 14296.812} C_VEL
LIN {X 0,Y 281.41,Z 1002.151,A -85,B 0,C 180,E1 14292.638,E2 14292.638} C_VEL
LIN {X 0,Y 283.447,Z 994.964,A -85,B 0,C 180,E1 14287.828,E2 14287.828} C_VEL
LIN {X 0,Y 286.239,Z 987.157,A -85,B 0,C 180,E1 14283.669,E2 14283.669} C_VEL
LIN {X 0,Y 290.533,Z 976.744,A -85,B 0,C 180,E1 14279.156,E2 14279.156} C_VEL
LIN {X 0,Y 295.628,Z 965.528,A -85,B 0,C 180,E1 14275.145,E2 14275.145} C_VEL
LIN {X 0,Y 301.866,Z 952.277,A -85,B 0,C 180,E1 14271.249,E2 14271.249} C_VEL
LIN {X 0,Y 308.906,Z 937.773,A -85,B 0,C 180,E1 14267.688,E2 14267.688} C_VEL
LIN {X 0,Y 316.094,Z 922.554,A -85,B 0,C 180,E1 14264.605,E2 14264.605} C_VEL
LIN {X 0,Y 324.252,Z 904.849,A -85,B 0,C 180,E1 14261.611,E2 14261.611} C_VEL
LIN {X 0,Y 331.683,Z 887.813,A -85,B 0,C 180,E1 14259.229,E2 14259.229} C_VEL
LIN {X 0,Y 339.646,Z 868.159,A -85,B 0,C 180,E1 14256.951,E2 14256.951} C_VEL
LIN {X 0,Y 346.335,Z 850.177,A -85,B 0,C 180,E1 14255.223,E2 14255.223} C_VEL
LIN {X 0,Y 353.333,Z 829.129,A -85,B 0,C 180,E1 14253.564,E2 14253.564} C_VEL
LIN {X 0,Y 359.158,Z 809.263,A -85,B 0,C 180,E1 14252.289,E2 14252.289} C_VEL
LIN {X 0,Y 364.577,Z 787.451,A -85,B 0,C 180,E1 14251.178,E2 14251.178} C_VEL
LIN {X 0,Y 368.727,Z 767.419,A -85,B 0,C 180,E1 14250.378,E2 14250.378} C_VEL
LIN {X 0,Y 372.517,Z 743.451,A -85,B 0,C 180,E1 14249.664,E2 14249.664} C_VEL
LIN {X 0,Y 374.92,Z 719.77,A -85,B 0,C 180,E1 14249.123,E2 14249.123} C_VEL
LIN {X 0,Y 388.944,Z 520.367,A -85,B 0,C 180,E1 14245.202,E2 14245.202} C_VEL
LIN {X 0,Y 383.481,Z 510.588,A -85,B 0,C 180,E1 14242.982,E2 14242.982} C_VEL
LIN {X 0,Y 377.989,Z 501.226,A -85,B 0,C 180,E1 14240.476,E2 14240.476} C_VEL
LIN {X 0,Y 372.687,Z 493.27,A -85,B 0,C 180,E1 14237.728,E2 14237.728} C_VEL
LIN {X 0,Y 368.459,Z 487.588,A -85,B 0,C 180,E1 14235.18,E2 14235.18} C_VEL
LIN {X 0,Y 365.186,Z 482.967,A -85,B 0,C 180,E1 14232.813,E2 14232.813} C_VEL
LIN {X 0,Y 362.273,Z 479.084,A -85,B 0,C 180,E1 14230.254,E2 14230.254} C_VEL
LIN {X 0,Y 361.622,Z 477.888,A -85,B 0,C 180,E1 14229.549,E2 14229.549} C_VEL
LIN {X 0,Y 358.542,Z 474.265,A -85,B 0,C 180,E1 14225.44,E2 14225.44} C_VEL
LIN {X 0,Y 357.807,Z 472.12,A -85,B 0,C 180,E1 14223.524,E2 14223.524} C_VEL
LIN {X 0,Y 357.596,Z 472.056,A -85,B 0,C 180,E1 14216.473,E2 14216.473} C_VEL
LIN {X 0,Y 357.979,Z 472.409,A -85,B 0,C 180,E1 14215.434,E2 14215.434} C_VEL
LIN {X 0,Y 359.874,Z 476.379,A -85,B 0,C 180,E1 14211.854,E2 14211.854} C_VEL
LIN {X 0,Y 361.909,Z 478.304,A -85,B 0,C 180,E1 14209.574,E2 14209.574} C_VEL
LIN {X 0,Y 364.681,Z 482.427,A -85,B 0,C 180,E1 14207.007,E2 14207.007} C_VEL
LIN {X 0,Y 365.979,Z 483.993,A -85,B 0,C 180,E1 14206.008,E2 14206.008} C_VEL
LIN {X 0,Y 369.872,Z 489.454,A -85,B 0,C 180,E1 14203.348,E2 14203.348} C_VEL
LIN {X 0,Y 373.935,Z 495.305,A -85,B 0,C 180,E1 14201.001,E2 14201.001} C_VEL
LIN {X 0,Y 379.223,Z 502.905,A -85,B 0,C 180,E1 14198.379,E2 14198.379} C_VEL
LIN {X 0,Y 385.89,Z 513.274,A -85,B 0,C 180,E1 14195.508,E2 14195.508} C_VEL
LIN {X 0,Y 388.848,Z 518.213,A -85,B 0,C 180,E1 14194.346,E2 14194.346} C_VEL
LIN {X 0,Y 374.67,Z 716.027,A -85,B 0,C 180,E1 14190.448,E2 14190.448} C_VEL
LIN {X 0,Y 371.576,Z 740.909,A -85,B 0,C 180,E1 14189.79,E2 14189.79} C_VEL
LIN {X 0,Y 368.076,Z 761.275,A -85,B 0,C 180,E1 14189.049,E2 14189.049} C_VEL
LIN {X 0,Y 363.136,Z 783.751,A -85,B 0,C 180,E1 14187.988,E2 14187.988} C_VEL
LIN {X 0,Y 358.16,Z 802.749,A -85,B 0,C 180,E1 14186.866,E2 14186.866} C_VEL
LIN {X 0,Y 351.803,Z 823.502,A -85,B 0,C 180,E1 14185.36,E2 14185.36} C_VEL
LIN {X 0,Y 345.649,Z 841.264,A -85,B 0,C 180,E1 14183.8,E2 14183.8} C_VEL
LIN {X 0,Y 337.821,Z 861.498,A -85,B 0,C 180,E1 14181.649,E2 14181.649} C_VEL
LIN {X 0,Y 330.191,Z 879.584,A -85,B 0,C 180,E1 14179.328,E2 14179.328} C_VEL
LIN {X 0,Y 322.343,Z 896.642,A -85,B 0,C 180,E1 14176.66,E2 14176.66} C_VEL
LIN {X 0,Y 314.536,Z 912.913,A -85,B 0,C 180,E1 14173.608,E2 14173.608} C_VEL
LIN {X 0,Y 307.612,Z 926.694,A -85,B 0,C 180,E1 14170.483,E2 14170.483} C_VEL
LIN {X 0,Y 300.363,Z 941.015,A -85,B 0,C 180,E1 14166.569,E2 14166.569} C_VEL
LIN {X 0,Y 294.785,Z 952.196,A -85,B 0,C 180,E1 14162.862,E2 14162.862} C_VEL
LIN {X 0,Y 289.784,Z 962.611,A -85,B 0,C 180,E1 14158.655,E2 14158.655} C_VEL
LIN {X 0,Y 285.971,Z 971.33,A -85,B 0,C 180,E1 14154.363,E2 14154.363} C_VEL
LIN {X 0,Y 283.133,Z 978.612,A -85,B 0,C 180,E1 14149.814,E2 14149.814} C_VEL
LIN {X 0,Y 281.375,Z 984.385,A -85,B 0,C 180,E1 14145.243,E2 14145.243} C_VEL
LIN {X 0,Y 280.425,Z 988.446,A -85,B 0,C 180,E1 14140.683,E2 14140.683} C_VEL
LIN {X 0,Y 280.103,Z 990.855,A -85,B 0,C 180,E1 14136.764,E2 14136.764} C_VEL
LIN {X 0,Y 279.994,Z 992.278,A -85,B 0,C 180,E1 14132.25,E2 14132.25} C_VEL
LIN {X 0,Y 279.988,Z 992.374,A -85,B 0,C 180,E1 14128.567,E2 14128.567} C_VEL
LIN {X 0,Y 280.042,Z 991.492,A -85,B 0,C 180,E1 14124.674,E2 14124.674} C_VEL
LIN {X 0,Y 280.337,Z 989.135,A -85,B 0,C 180,E1 14120.143,E2 14120.143} C_VEL
LIN {X 0,Y 281.081,Z 985.483,A -85,B 0,C 180,E1 14115.793,E2 14115.793} C_VEL
LIN {X 0,Y 282.798,Z 979.632,A -85,B 0,C 180,E1 14110.805,E2 14110.805} C_VEL
LIN {X 0,Y 285.156,Z 973.271,A -85,B 0,C 180,E1 14106.66,E2 14106.66} C_VEL
LIN {X 0,Y 289.079,Z 964.155,A -85,B 0,C 180,E1 14101.943,E2 14101.943} C_VEL
LIN {X 0,Y 293.904,Z 954.075,A -85,B 0,C 180,E1 14097.72,E2 14097.72} C_VEL
LIN {X 0,Y 297.809,Z 946.22,A -85,B 0,C 180,E1 14094.951,E2 14094.951} C_VEL
LIN {X 0,Y 298.826,Z 942.507,A -85,B 0,C 180,E1 14093.654,E2 14093.654} C_VEL
LIN {X 0,Y 298.911,Z 932.963,A -85,B 0,C 180,E1 14090.014,E2 14090.014} C_VEL
LIN {X 0,Y 300.209,Z 929.348,A -85,B 0,C 180,E1 14088.975,E2 14088.975} C_VEL
LIN {X 0,Y 307.663,Z 915.112,A -85,B 0,C 180,E1 14085.641,E2 14085.641} C_VEL
LIN {X 0,Y 316.127,Z 898.372,A -85,B 0,C 180,E1 14082.401,E2 14082.401} C_VEL
LIN {X 0,Y 323.966,Z 882.051,A -85,B 0,C 180,E1 14079.789,E2 14079.789} C_VEL
LIN {X 0,Y 331.823,Z 864.337,A -85,B 0,C 180,E1 14077.448,E2 14077.448} C_VEL
LIN {X 0,Y 339.286,Z 846.136,A -85,B 0,C 180,E1 14075.437,E2 14075.437} C_VEL
LIN {X 0,Y 346.471,Z 826.352,A -85,B 0,C 180,E1 14073.648,E2 14073.648} C_VEL
LIN {X 0,Y 353.027,Z 806.177,A -85,B 0,C 180,E1 14072.14,E2 14072.14} C_VEL
LIN {X 0,Y 358.447,Z 786.342,A -85,B 0,C 180,E1 14070.946,E2 14070.946} C_VEL
LIN {X 0,Y 363.359,Z 765.41,A -85,B 0,C 180,E1 14069.923,E2 14069.923} C_VEL
LIN {X 0,Y 367.397,Z 743.13,A -85,B 0,C 180,E1 14069.092,E2 14069.092} C_VEL
LIN {X 0,Y 370.571,Z 719.836,A -85,B 0,C 180,E1 14068.453,E2 14068.453} C_VEL
LIN {X 0,Y 376.717,Z 637.839,A -85,B 0,C 180,E1 14066.816,E2 14066.816} C_VEL
LIN {X 0,Y 385.182,Z 522.664,A -85,B 0,C 180,E1 14064.54,E2 14064.54} C_VEL
LIN {X 0,Y 377.963,Z 511.295,A -85,B 0,C 180,E1 14061.412,E2 14061.412} C_VEL
LIN {X 0,Y 372.884,Z 503.698,A -85,B 0,C 180,E1 14058.851,E2 14058.851} C_VEL
LIN {X 0,Y 369.888,Z 499.33,A -85,B 0,C 180,E1 14057.136,E2 14057.136} C_VEL
LIN {X 0,Y 367.178,Z 495.383,A -85,B 0,C 180,E1 14055.397,E2 14055.397} C_VEL
LIN {X 0,Y 363.991,Z 490.734,A -85,B 0,C 180,E1 14053.018,E2 14053.018} C_VEL
LIN {X 0,Y 361.016,Z 486.669,A -85,B 0,C 180,E1 14050.291,E2 14050.291} C_VEL
LIN {X 0,Y 360.382,Z 485.646,A -85,B 0,C 180,E1 14049.583,E2 14049.583} C_VEL
LIN {X 0,Y 357.457,Z 481.866,A -85,B 0,C 180,E1 14045.297,E2 14045.297} C_VEL
LIN {X 0,Y 356.935,Z 480.074,A -85,B 0,C 180,E1 14043.694,E2 14043.694} C_VEL
LIN {X 0,Y 356.99,Z 480.128,A -85,B 0,C 180,E1 14036.628,E2 14036.628} C_VEL
LIN {X 0,Y 358.8,Z 484.238,A -85,B 0,C 180,E1 14032.797,E2 14032.797} C_VEL
LIN {X 0,Y 360.809,Z 486.227,A -85,B 0,C 180,E1 14030.429,E2 14030.429} C_VEL
LIN {X 0,Y 363.586,Z 490.438,A -85,B 0,C 180,E1 14027.776,E2 14027.776} C_VEL
LIN {X 0,Y 364.754,Z 491.896,A -85,B 0,C 180,E1 14026.849,E2 14026.849} C_VEL
LIN {X 0,Y 368.55,Z 497.393,A -85,B 0,C 180,E1 14024.178,E2 14024.178} C_VEL
LIN {X 0,Y 372.205,Z 502.676,A -85,B 0,C 180,E1 14022.006,E2 14022.006} C_VEL
LIN {X 0,Y 376.508,Z 509.156,A -85,B 0,C 180,E1 14019.764,E2 14019.764} C_VEL
LIN {X 0,Y 383.139,Z 520.838,A -85,B 0,C 180,E1 14016.712,E2 14016.712} C_VEL
LIN {X 0,Y 385.321,Z 525.095,A -85,B 0,C 180,E1 14015.789,E2 14015.789} C_VEL
LIN {X 0,Y 370.539,Z 726.52,A -85,B 0,C 180,E1 14011.821,E2 14011.821} C_VEL
LIN {X 0,Y 367.765,Z 750.071,A -85,B 0,C 180,E1 14011.253,E2 14011.253} C_VEL
LIN {X 0,Y 363.659,Z 772.776,A -85,B 0,C 180,E1 14010.523,E2 14010.523} C_VEL
LIN {X 0,Y 358.43,Z 795.852,A -85,B 0,C 180,E1 14009.528,E2 14009.528} C_VEL
LIN {X 0,Y 352.914,Z 815.995,A -85,B 0,C 180,E1 14008.412,E2 14008.412} C_VEL
LIN {X 0,Y 345.716,Z 838.564,A -85,B 0,C 180,E1 14006.844,E2 14006.844} C_VEL
LIN {X 0,Y 338.634,Z 858.203,A -85,B 0,C 180,E1 14005.159,E2 14005.159} C_VEL
LIN {X 0,Y 330.817,Z 877.558,A -85,B 0,C 180,E1 14003.12,E2 14003.12} C_VEL
LIN {X 0,Y 322.738,Z 896.194,A -85,B 0,C 180,E1 14000.753,E2 14000.753} C_VEL
LIN {X 0,Y 314.55,Z 913.578,A -85,B 0,C 180,E1 13998.051,E2 13998.051} C_VEL
LIN {X 0,Y 306.181,Z 930.645,A -85,B 0,C 180,E1 13994.853,E2 13994.853} C_VEL
LIN {X 0,Y 299.129,Z 944.622,A -85,B 0,C 180,E1 13991.69,E2 13991.69} C_VEL
LIN {X 0,Y 291.934,Z 958.864,A -85,B 0,C 180,E1 13987.807,E2 13987.807} C_VEL
LIN {X 0,Y 285.937,Z 971.103,A -85,B 0,C 180,E1 13983.775,E2 13983.775} C_VEL
LIN {X 0,Y 280.905,Z 981.891,A -85,B 0,C 180,E1 13979.416,E2 13979.416} C_VEL
LIN {X 0,Y 277.153,Z 991.022,A -85,B 0,C 180,E1 13974.964,E2 13974.964} C_VEL
LIN {X 0,Y 274.471,Z 998.636,A -85,B 0,C 180,E1 13970.245,E2 13970.245} C_VEL
LIN {X 0,Y 272.872,Z 1004.715,A -85,B 0,C 180,E1 13965.491,E2 13965.491} C_VEL
LIN {X 0,Y 272.173,Z 1008.839,A -85,B 0,C 180,E1 13961.012,E2 13961.012} C_VEL
LIN {X 0,Y 271.972,Z 1011.438,A -85,B 0,C 180,E1 13956.968,E2 13956.968} C_VEL
LIN {X 0,Y 271.976,Z 1012.941,A -85,B 0,C 180,E1 13952.529,E2 13952.529} C_VEL
LIN {X 0,Y 271.987,Z 1013.085,A -85,B 0,C 180,E1 13948.737,E2 13948.737} C_VEL
LIN {X 0,Y 271.969,Z 1012.226,A -85,B 0,C 180,E1 13944.939,E2 13944.939} C_VEL
LIN {X 0,Y 272.069,Z 1009.992,A -85,B 0,C 180,E1 13940.483,E2 13940.483} C_VEL
LIN {X 0,Y 272.579,Z 1006.188,A -85,B 0,C 180,E1 13935.992,E2 13935.992} C_VEL
LIN {X 0,Y 273.771,Z 1001.05,A -85,B 0,C 180,E1 13931.477,E2 13931.477} C_VEL
LIN {X 0,Y 276.027,Z 993.924,A -85,B 0,C 180,E1 13926.748,E2 13926.748} C_VEL
LIN {X 0,Y 279.525,Z 985.162,A -85,B 0,C 180,E1 13922.062,E2 13922.062} C_VEL
LIN {X 0,Y 284.175,Z 974.705,A -85,B 0,C 180,E1 13917.61,E2 13917.61} C_VEL
LIN {X 0,Y 290.302,Z 962.067,A -85,B 0,C 180,E1 13913.187,E2 13913.187} C_VEL
LIN {X 0,Y 296.473,Z 949.818,A -85,B 0,C 180,E1 13909.651,E2 13909.651} C_VEL
LIN {X 0,Y 304.008,Z 934.878,A -85,B 0,C 180,E1 13906.062,E2 13906.062} C_VEL
LIN {X 0,Y 311.645,Z 919.521,A -85,B 0,C 180,E1 13902.996,E2 13902.996} C_VEL
LIN {X 0,Y 319.83,Z 902.286,A -85,B 0,C 180,E1 13900.159,E2 13900.159} C_VEL
LIN {X 0,Y 327.877,Z 884.484,A -85,B 0,C 180,E1 13897.713,E2 13897.713} C_VEL
LIN {X 0,Y 335.635,Z 865.62,A -85,B 0,C 180,E1 13895.594,E2 13895.594} C_VEL
LIN {X 0,Y 343.133,Z 845.881,A -85,B 0,C 180,E1 13893.752,E2 13893.752} C_VEL
LIN {X 0,Y 349.84,Z 825.781,A -85,B 0,C 180,E1 13892.234,E2 13892.234} C_VEL
LIN {X 0,Y 356.196,Z 804.138,A -85,B 0,C 180,E1 13890.909,E2 13890.909} C_VEL
LIN {X 0,Y 361.315,Z 783.348,A -85,B 0,C 180,E1 13889.91,E2 13889.91} C_VEL
LIN {X 0,Y 366.057,Z 759.677,A -85,B 0,C 180,E1 13889.041,E2 13889.041} C_VEL
LIN {X 0,Y 369.33,Z 737.516,A -85,B 0,C 180,E1 13888.435,E2 13888.435} C_VEL
LIN {X 0,Y 372.122,Z 704.51,A -85,B 0,C 180,E1 13887.741,E2 13887.741} C_VEL
LIN {X 0,Y 385.222,Z 524.801,A -85,B 0,C 180,E1 13884.21,E2 13884.21} C_VEL
LIN {X 0,Y 378.858,Z 513.394,A -85,B 0,C 180,E1 13881.439,E2 13881.439} C_VEL
LIN {X 0,Y 374.424,Z 505.996,A -85,B 0,C 180,E1 13879.256,E2 13879.256} C_VEL
LIN {X 0,Y 370.118,Z 499.715,A -85,B 0,C 180,E1 13876.882,E2 13876.882} C_VEL
LIN {X 0,Y 367.019,Z 495.275,A -85,B 0,C 180,E1 13874.918,E2 13874.918} C_VEL
LIN {X 0,Y 363.814,Z 490.674,A -85,B 0,C 180,E1 13872.539,E2 13872.539} C_VEL
LIN {X 0,Y 360.912,Z 486.628,A -85,B 0,C 180,E1 13869.89,E2 13869.89} C_VEL
LIN {X 0,Y 360.191,Z 485.563,A -85,B 0,C 180,E1 13869.104,E2 13869.104} C_VEL
LIN {X 0,Y 357.406,Z 481.969,A -85,B 0,C 180,E1 13865.136,E2 13865.136} C_VEL
LIN {X 0,Y 356.771,Z 480.041,A -85,B 0,C 180,E1 13863.374,E2 13863.374} C_VEL
LIN {X 0,Y 356.678,Z 480.015,A -85,B 0,C 180,E1 13856.303,E2 13856.303} C_VEL
LIN {X 0,Y 356.958,Z 480.443,A -85,B 0,C 180,E1 13855.501,E2 13855.501} C_VEL
LIN {X 0,Y 359.021,Z 484.536,A -85,B 0,C 180,E1 13851.673,E2 13851.673} C_VEL
LIN {X 0,Y 360.699,Z 486.156,A -85,B 0,C 180,E1 13849.781,E2 13849.781} C_VEL
LIN {X 0,Y 363.517,Z 490.326,A -85,B 0,C 180,E1 13847.127,E2 13847.127} C_VEL
LIN {X 0,Y 364.685,Z 491.892,A -85,B 0,C 180,E1 13846.2,E2 13846.2} C_VEL
LIN {X 0,Y 368.401,Z 497.205,A -85,B 0,C 180,E1 13843.604,E2 13843.604} C_VEL
LIN {X 0,Y 372.193,Z 502.772,A -85,B 0,C 180,E1 13841.356,E2 13841.356} C_VEL
LIN {X 0,Y 377.37,Z 510.432,A -85,B 0,C 180,E1 13838.716,E2 13838.716} C_VEL
LIN {X 0,Y 384.01,Z 520.973,A -85,B 0,C 180,E1 13835.789,E2 13835.789} C_VEL
LIN {X 0,Y 385.116,Z 522.992,A -85,B 0,C 180,E1 13835.332,E2 13835.332} C_VEL
LIN {X 0,Y 370.693,Z 717.418,A -85,B 0,C 180,E1 13831.5,E2 13831.5} C_VEL
LIN {X 0,Y 367.536,Z 741.691,A -85,B 0,C 180,E1 13830.854,E2 13830.854} C_VEL
LIN {X 0,Y 363.894,Z 762.235,A -85,B 0,C 180,E1 13830.106,E2 13830.106} C_VEL
LIN {X 0,Y 358.939,Z 784.061,A -85,B 0,C 180,E1 13829.077,E2 13829.077} C_VEL
LIN {X 0,Y 353.816,Z 803.059,A -85,B 0,C 180,E1 13827.959,E2 13827.959} C_VEL
LIN {X 0,Y 347.124,Z 824.228,A -85,B 0,C 180,E1 13826.424,E2 13826.424} C_VEL
LIN {X 0,Y 340.623,Z 842.377,A -85,B 0,C 180,E1 13824.825,E2 13824.825} C_VEL
LIN {X 0,Y 332.826,Z 861.808,A -85,B 0,C 180,E1 13822.75,E2 13822.75} C_VEL
LIN {X 0,Y 325.186,Z 879.293,A -85,B 0,C 180,E1 13820.503,E2 13820.503} C_VEL
LIN {X 0,Y 317.007,Z 896.454,A -85,B 0,C 180,E1 13817.826,E2 13817.826} C_VEL
LIN {X 0,Y 309.066,Z 912.393,A -85,B 0,C 180,E1 13814.843,E2 13814.843} C_VEL
LIN {X 0,Y 301.471,Z 926.827,A -85,B 0,C 180,E1 13811.547,E2 13811.547} C_VEL
LIN {X 0,Y 294.093,Z 940.705,A -85,B 0,C 180,E1 13807.726,E2 13807.726} C_VEL
LIN {X 0,Y 288.156,Z 951.947,A -85,B 0,C 180,E1 13803.957,E2 13803.957} C_VEL
LIN {X 0,Y 282.56,Z 962.923,A -85,B 0,C 180,E1 13799.459,E2 13799.459} C_VEL
LIN {X 0,Y 278.321,Z 972.033,A -85,B 0,C 180,E1 13794.851,E2 13794.851} C_VEL
LIN {X 0,Y 275.32,Z 979.214,A -85,B 0,C 180,E1 13790.179,E2 13790.179} C_VEL
LIN {X 0,Y 273.453,Z 984.9,A -85,B 0,C 180,E1 13785.479,E2 13785.479} C_VEL
LIN {X 0,Y 272.481,Z 988.75,A -85,B 0,C 180,E1 13780.998,E2 13780.998} C_VEL
LIN {X 0,Y 272.118,Z 991.157,A -85,B 0,C 180,E1 13776.963,E2 13776.963} C_VEL
LIN {X 0,Y 271.999,Z 992.557,A -85,B 0,C 180,E1 13772.527,E2 13772.527} C_VEL
LIN {X 0,Y 271.994,Z 992.674,A -85,B 0,C 180,E1 13768.525,E2 13768.525} C_VEL
LIN {X 0,Y 272.055,Z 991.793,A -85,B 0,C 180,E1 13764.517,E2 13764.517} C_VEL
LIN {X 0,Y 272.375,Z 989.438,A -85,B 0,C 180,E1 13759.852,E2 13759.852} C_VEL
LIN {X 0,Y 273.144,Z 985.987,A -85,B 0,C 180,E1 13755.588,E2 13755.588} C_VEL
LIN {X 0,Y 274.868,Z 980.525,A -85,B 0,C 180,E1 13750.671,E2 13750.671} C_VEL
LIN {X 0,Y 277.458,Z 973.922,A -85,B 0,C 180,E1 13746.198,E2 13746.198} C_VEL
LIN {X 0,Y 281.731,Z 964.64,A -85,B 0,C 180,E1 13741.235,E2 13741.235} C_VEL
LIN {X 0,Y 286.662,Z 954.886,A -85,B 0,C 180,E1 13737.039,E2 13737.039} C_VEL
LIN {X 0,Y 292.646,Z 943.464,A -85,B 0,C 180,E1 13733.04,E2 13733.04} C_VEL
LIN {X 0,Y 299.687,Z 930.37,A -85,B 0,C 180,E1 13729.232,E2 13729.232} C_VEL
LIN {X 0,Y 300.209,Z 929.348,A -85,B 0,C 180,E1 13728.975,E2 13728.975} C_VEL
LIN {X 0,Y 301.708,Z 925.069,A -85,B 0,C 180,E1 13727.775,E2 13727.775} C_VEL
LIN {X 0,Y 303.142,Z 914.042,A -85,B 0,C 180,E1 13724.345,E2 13724.345} C_VEL
LIN {X 0,Y 304.76,Z 909.96,A -85,B 0,C 180,E1 13723.403,E2 13723.403} C_VEL
LIN {X 0,Y 312.589,Z 894.89,A -85,B 0,C 180,E1 13720.631,E2 13720.631} C_VEL
LIN {X 0,Y 321.547,Z 876.49,A -85,B 0,C 180,E1 13717.839,E2 13717.839} C_VEL
LIN {X 0,Y 329.432,Z 858.984,A -85,B 0,C 180,E1 13715.644,E2 13715.644} C_VEL
LIN {X 0,Y 337.124,Z 839.97,A -85,B 0,C 180,E1 13713.684,E2 13713.684} C_VEL
LIN {X 0,Y 344.281,Z 820.389,A -85,B 0,C 180,E1 13712.012,E2 13712.012} C_VEL
LIN {X 0,Y 350.74,Z 799.75,A -85,B 0,C 180,E1 13710.591,E2 13710.591} C_VEL
LIN {X 0,Y 356.554,Z 778.232,A -85,B 0,C 180,E1 13709.39,E2 13709.39} C_VEL
LIN {X 0,Y 361.294,Z 756.226,A -85,B 0,C 180,E1 13708.438,E2 13708.438} C_VEL
LIN {X 0,Y 365.188,Z 733.033,A -85,B 0,C 180,E1 13707.682,E2 13707.682} C_VEL
LIN {X 0,Y 367.677,Z 711.037,A -85,B 0,C 180,E1 13707.159,E2 13707.159} C_VEL
LIN {X 0,Y 381.594,Z 527.667,A -85,B 0,C 180,E1 13703.552,E2 13703.552} C_VEL
LIN {X 0,Y 375.161,Z 517.182,A -85,B 0,C 180,E1 13700.598,E2 13700.598} C_VEL
LIN {X 0,Y 369.161,Z 508.018,A -85,B 0,C 180,E1 13697.334,E2 13697.334} C_VEL
LIN {X 0,Y 365.525,Z 502.806,A -85,B 0,C 180,E1 13694.981,E2 13694.981} C_VEL
LIN {X 0,Y 362.438,Z 498.252,A -85,B 0,C 180,E1 13692.588,E2 13692.588} C_VEL
LIN {X 0,Y 359.609,Z 494.07,A -85,B 0,C 180,E1 13689.846,E2 13689.846} C_VEL
LIN {X 0,Y 356.231,Z 489.189,A -85,B 0,C 180,E1 13684.669,E2 13684.669} C_VEL
LIN {X 0,Y 355.905,Z 488,A -85,B 0,C 180,E1 13683.544,E2 13683.544} C_VEL
LIN {X 0,Y 355.959,Z 488.035,A -85,B 0,C 180,E1 13676.78,E2 13676.78} C_VEL
LIN {X 0,Y 357.712,Z 492.115,A -85,B 0,C 180,E1 13672.936,E2 13672.936} C_VEL
LIN {X 0,Y 359.606,Z 494.074,A -85,B 0,C 180,E1 13670.639,E2 13670.639} C_VEL
LIN {X 0,Y 362.424,Z 498.331,A -85,B 0,C 180,E1 13667.897,E2 13667.897} C_VEL
LIN {X 0,Y 363.655,Z 500.122,A -85,B 0,C 180,E1 13666.89,E2 13666.89} C_VEL
LIN {X 0,Y 366.973,Z 504.942,A -85,B 0,C 180,E1 13664.514,E2 13664.514} C_VEL
LIN {X 0,Y 370.48,Z 510.139,A -85,B 0,C 180,E1 13662.366,E2 13662.366} C_VEL
LIN {X 0,Y 374.616,Z 516.547,A -85,B 0,C 180,E1 13660.146,E2 13660.146} C_VEL
LIN {X 0,Y 381.024,Z 528.167,A -85,B 0,C 180,E1 13657.106,E2 13657.106} C_VEL
LIN {X 0,Y 381.704,Z 529.746,A -85,B 0,C 180,E1 13656.796,E2 13656.796} C_VEL
LIN {X 0,Y 366.663,Z 727.781,A -85,B 0,C 180,E1 13652.896,E2 13652.896} C_VEL
LIN {X 0,Y 363.603,Z 751.845,A -85,B 0,C 180,E1 13652.305,E2 13652.305} C_VEL
LIN {X 0,Y 359.514,Z 773.682,A -85,B 0,C 180,E1 13651.598,E2 13651.598} C_VEL
LIN {X 0,Y 354.042,Z 796.848,A -85,B 0,C 180,E1 13650.592,E2 13650.592} C_VEL
LIN {X 0,Y 348.254,Z 817.288,A -85,B 0,C 180,E1 13649.455,E2 13649.455} C_VEL
LIN {X 0,Y 340.989,Z 839.171,A -85,B 0,C 180,E1 13647.922,E2 13647.922} C_VEL
LIN {X 0,Y 333.393,Z 859.518,A -85,B 0,C 180,E1 13646.165,E2 13646.165} C_VEL
LIN {X 0,Y 325.232,Z 878.852,A -85,B 0,C 180,E1 13644.095,E2 13644.095} C_VEL
LIN {X 0,Y 316.64,Z 897.741,A -85,B 0,C 180,E1 13641.641,E2 13641.641} C_VEL
LIN {X 0,Y 308.534,Z 914.296,A -85,B 0,C 180,E1 13639.025,E2 13639.025} C_VEL
LIN {X 0,Y 299.852,Z 931.193,A -85,B 0,C 180,E1 13635.795,E2 13635.795} C_VEL
LIN {X 0,Y 292.513,Z 945.094,A -85,B 0,C 180,E1 13632.588,E2 13632.588} C_VEL
LIN {X 0,Y 285.001,Z 959.199,A -85,B 0,C 180,E1 13628.639,E2 13628.639} C_VEL
LIN {X 0,Y 278.713,Z 971.375,A -85,B 0,C 180,E1 13624.524,E2 13624.524} C_VEL
LIN {X 0,Y 273.422,Z 982.049,A -85,B 0,C 180,E1 13620.062,E2 13620.062} C_VEL
LIN {X 0,Y 269.3,Z 991.446,A -85,B 0,C 180,E1 13615.273,E2 13615.273} C_VEL
LIN {X 0,Y 266.62,Z 998.64,A -85,B 0,C 180,E1 13610.639,E2 13610.639} C_VEL
LIN {X 0,Y 264.875,Z 1004.816,A -85,B 0,C 180,E1 13605.545,E2 13605.545} C_VEL
LIN {X 0,Y 264.182,Z 1008.701,A -85,B 0,C 180,E1 13601.128,E2 13601.128} C_VEL
LIN {X 0,Y 263.983,Z 1011.487,A -85,B 0,C 180,E1 13596.524,E2 13596.524} C_VEL
LIN {X 0,Y 263.991,Z 1012.69,A -85,B 0,C 180,E1 13592.171,E2 13592.171} C_VEL
LIN {X 0,Y 263.995,Z 1012.761,A -85,B 0,C 180,E1 13588.482,E2 13588.482} C_VEL
LIN {X 0,Y 263.971,Z 1011.853,A -85,B 0,C 180,E1 13584.568,E2 13584.568} C_VEL
LIN {X 0,Y 264.098,Z 1009.426,A -85,B 0,C 180,E1 13579.844,E2 13579.844} C_VEL
LIN {X 0,Y 264.69,Z 1005.666,A -85,B 0,C 180,E1 13575.342,E2 13575.342} C_VEL
LIN {X 0,Y 266.135,Z 1000.189,A -85,B 0,C 180,E1 13570.469,E2 13570.469} C_VEL
LIN {X 0,Y 268.703,Z 992.883,A -85,B 0,C 180,E1 13565.608,E2 13565.608} C_VEL
LIN {X 0,Y 272.574,Z 983.908,A -85,B 0,C 180,E1 13560.804,E2 13560.804} C_VEL
LIN {X 0,Y 277.329,Z 974.004,A -85,B 0,C 180,E1 13556.527,E2 13556.527} C_VEL
LIN {X 0,Y 283.962,Z 961.103,A -85,B 0,C 180,E1 13551.967,E2 13551.967} C_VEL
LIN {X 0,Y 290.91,Z 948.073,A -85,B 0,C 180,E1 13548.188,E2 13548.188} C_VEL
LIN {X 0,Y 298.718,Z 933.244,A -85,B 0,C 180,E1 13544.66,E2 13544.66} C_VEL
LIN {X 0,Y 307.024,Z 917.295,A -85,B 0,C 180,E1 13541.503,E2 13541.503} C_VEL
LIN {X 0,Y 315.345,Z 900.284,A -85,B 0,C 180,E1 13538.75,E2 13538.75} C_VEL
LIN {X 0,Y 323.946,Z 881.672,A -85,B 0,C 180,E1 13536.25,E2 13536.25} C_VEL
LIN {X 0,Y 331.785,Z 863.174,A -85,B 0,C 180,E1 13534.215,E2 13534.215} C_VEL
LIN {X 0,Y 340.048,Z 841.57,A -85,B 0,C 180,E1 13532.278,E2 13532.278} C_VEL
LIN {X 0,Y 346.891,Z 821.422,A -85,B 0,C 180,E1 13530.814,E2 13530.814} C_VEL
LIN {X 0,Y 352.981,Z 800.444,A -85,B 0,C 180,E1 13529.599,E2 13529.599} C_VEL
LIN {X 0,Y 358.353,Z 778.795,A -85,B 0,C 180,E1 13528.603,E2 13528.603} C_VEL
LIN {X 0,Y 362.814,Z 755.804,A -85,B 0,C 180,E1 13527.819,E2 13527.819} C_VEL
LIN {X 0,Y 366.156,Z 732.109,A -85,B 0,C 180,E1 13527.206,E2 13527.206} C_VEL
LIN {X 0,Y 374.145,Z 627.325,A -85,B 0,C 180,E1 13525.121,E2 13525.121} C_VEL
LIN {X 0,Y 381.567,Z 529.291,A -85,B 0,C 180,E1 13523.185,E2 13523.185} C_VEL
LIN {X 0,Y 374.848,Z 517.073,A -85,B 0,C 180,E1 13520.045,E2 13520.045} C_VEL
LIN {X 0,Y 370.801,Z 510.73,A -85,B 0,C 180,E1 13517.902,E2 13517.902} C_VEL
LIN {X 0,Y 368.128,Z 506.756,A -85,B 0,C 180,E1 13516.326,E2 13516.326} C_VEL
LIN {X 0,Y 365.362,Z 502.693,A -85,B 0,C 180,E1 13514.501,E2 13514.501} C_VEL
LIN {X 0,Y 362.451,Z 498.38,A -85,B 0,C 180,E1 13512.263,E2 13512.263} C_VEL
LIN {X 0,Y 359.565,Z 494.172,A -85,B 0,C 180,E1 13509.523,E2 13509.523} C_VEL
LIN {X 0,Y 358.644,Z 493.106,A -85,B 0,C 180,E1 13508.497,E2 13508.497} C_VEL
LIN {X 0,Y 356.216,Z 489.479,A -85,B 0,C 180,E1 13504.669,E2 13504.669} C_VEL
LIN {X 0,Y 355.738,Z 487.96,A -85,B 0,C 180,E1 13503.222,E2 13503.222} C_VEL
LIN {X 0,Y 355.764,Z 487.972,A -85,B 0,C 180,E1 13496.132,E2 13496.132} C_VEL
LIN {X 0,Y 358.435,Z 492.923,A -85,B 0,C 180,E1 13491.174,E2 13491.174} C_VEL
LIN {X 0,Y 359.494,Z 494.004,A -85,B 0,C 180,E1 13489.989,E2 13489.989} C_VEL
LIN {X 0,Y 362.354,Z 498.225,A -85,B 0,C 180,E1 13487.247,E2 13487.247} C_VEL
LIN {X 0,Y 366.711,Z 504.569,A -85,B 0,C 180,E1 13484.015,E2 13484.015} C_VEL
LIN {X 0,Y 370.597,Z 510.44,A -85,B 0,C 180,E1 13481.64,E2 13481.64} C_VEL
LIN {X 0,Y 375.605,Z 518.078,A -85,B 0,C 180,E1 13479.02,E2 13479.02} C_VEL
LIN {X 0,Y 381.503,Z 527.72,A -85,B 0,C 180,E1 13476.337,E2 13476.337} C_VEL
LIN {X 0,Y 366.873,Z 718.492,A -85,B 0,C 180,E1 13472.582,E2 13472.582} C_VEL
LIN {X 0,Y 363.646,Z 742.356,A -85,B 0,C 180,E1 13471.945,E2 13471.945} C_VEL
LIN {X 0,Y 359.838,Z 763.195,A -85,B 0,C 180,E1 13471.188,E2 13471.188} C_VEL
LIN {X 0,Y 354.875,Z 784.371,A -85,B 0,C 180,E1 13470.19,E2 13470.19} C_VEL
LIN {X 0,Y 349.605,Z 803.369,A -85,B 0,C 180,E1 13469.08,E2 13469.08} C_VEL
LIN {X 0,Y 342.898,Z 824.024,A -85,B 0,C 180,E1 13467.593,E2 13467.593} C_VEL
LIN {X 0,Y 336.202,Z 842.178,A -85,B 0,C 180,E1 13466.006,E2 13466.006} C_VEL
LIN {X 0,Y 327.958,Z 862.119,A -85,B 0,C 180,E1 13463.883,E2 13463.883} C_VEL
LIN {X 0,Y 320.048,Z 879.604,A -85,B 0,C 180,E1 13461.633,E2 13461.633} C_VEL
LIN {X 0,Y 311.556,Z 896.765,A -85,B 0,C 180,E1 13458.945,E2 13458.945} C_VEL
LIN {X 0,Y 303.183,Z 912.872,A -85,B 0,C 180,E1 13455.905,E2 13455.905} C_VEL
LIN {X 0,Y 295.34,Z 927.14,A -85,B 0,C 180,E1 13452.61,E2 13452.61} C_VEL
LIN {X 0,Y 287.592,Z 941.018,A -85,B 0,C 180,E1 13448.735,E2 13448.735} C_VEL
LIN {X 0,Y 281.12,Z 952.652,A -85,B 0,C 180,E1 13444.755,E2 13444.755} C_VEL
LIN {X 0,Y 275.229,Z 963.537,A -85,B 0,C 180,E1 13440.161,E2 13440.161} C_VEL
LIN {X 0,Y 270.863,Z 972.344,A -85,B 0,C 180,E1 13435.584,E2 13435.584} C_VEL
LIN {X 0,Y 267.637,Z 979.523,A -85,B 0,C 180,E1 13430.785,E2 13430.785} C_VEL
LIN {X 0,Y 265.6,Z 985.207,A -85,B 0,C 180,E1 13425.948,E2 13425.948} C_VEL
LIN {X 0,Y 264.546,Z 989.054,A -85,B 0,C 180,E1 13421.332,E2 13421.332} C_VEL
LIN {X 0,Y 264.134,Z 991.459,A -85,B 0,C 180,E1 13417.175,E2 13417.175} C_VEL
LIN {X 0,Y 264.004,Z 992.857,A -85,B 0,C 180,E1 13412.604,E2 13412.604} C_VEL
LIN {X 0,Y 264.001,Z 992.974,A -85,B 0,C 180,E1 13408.48,E2 13408.48} C_VEL
LIN {X 0,Y 264.068,Z 992.093,A -85,B 0,C 180,E1 13404.35,E2 13404.35} C_VEL
LIN {X 0,Y 264.425,Z 989.683,A -85,B 0,C 180,E1 13399.461,E2 13399.461} C_VEL
LIN {X 0,Y 265.327,Z 986.092,A -85,B 0,C 180,E1 13394.93,E2 13394.93} C_VEL
LIN {X 0,Y 267.251,Z 980.538,A -85,B 0,C 180,E1 13389.869,E2 13389.869} C_VEL
LIN {X 0,Y 269.943,Z 974.229,A -85,B 0,C 180,E1 13385.493,E2 13385.493} C_VEL
LIN {X 0,Y 274.379,Z 965.219,A -85,B 0,C 180,E1 13380.534,E2 13380.534} C_VEL
LIN {X 0,Y 279.463,Z 955.697,A -85,B 0,C 180,E1 13376.324,E2 13376.324} C_VEL
LIN {X 0,Y 286.072,Z 943.772,A -85,B 0,C 180,E1 13372.042,E2 13372.042} C_VEL
LIN {X 0,Y 293.375,Z 930.851,A -85,B 0,C 180,E1 13368.226,E2 13368.226} C_VEL
LIN {X 0,Y 301.294,Z 916.38,A -85,B 0,C 180,E1 13364.757,E2 13364.757} C_VEL
LIN {X 0,Y 304.76,Z 909.96,A -85,B 0,C 180,E1 13363.403,E2 13363.403} C_VEL
LIN {X 0,Y 306.622,Z 905.171,A -85,B 0,C 180,E1 13362.317,E2 13362.317} C_VEL
LIN {X 0,Y 309.129,Z 892.687,A -85,B 0,C 180,E1 13359.156,E2 13359.156} C_VEL
LIN {X 0,Y 310.954,Z 888.116,A -85,B 0,C 180,E1 13358.321,E2 13358.321} C_VEL
LIN {X 0,Y 319.501,Z 870.782,A -85,B 0,C 180,E1 13355.861,E2 13355.861} C_VEL
LIN {X 0,Y 327.933,Z 851.832,A -85,B 0,C 180,E1 13353.666,E2 13353.666} C_VEL
LIN {X 0,Y 335.816,Z 832.354,A -85,B 0,C 180,E1 13351.803,E2 13351.803} C_VEL
LIN {X 0,Y 342.689,Z 812.774,A -85,B 0,C 180,E1 13350.283,E2 13350.283} C_VEL
LIN {X 0,Y 349.19,Z 791.633,A -85,B 0,C 180,E1 13348.941,E2 13348.941} C_VEL
LIN {X 0,Y 354.453,Z 770.861,A -85,B 0,C 180,E1 13347.895,E2 13347.895} C_VEL
LIN {X 0,Y 359.36,Z 746.763,A -85,B 0,C 180,E1 13346.959,E2 13346.959} C_VEL
LIN {X 0,Y 362.685,Z 724.74,A -85,B 0,C 180,E1 13346.335,E2 13346.335} C_VEL
LIN {X 0,Y 365.674,Z 691.603,A -85,B 0,C 180,E1 13345.645,E2 13345.645} C_VEL
LIN {X 0,Y 378.09,Z 532.527,A -85,B 0,C 180,E1 13342.527,E2 13342.527} C_VEL
LIN {X 0,Y 372.338,Z 523.199,A -85,B 0,C 180,E1 13339.736,E2 13339.736} C_VEL
LIN {X 0,Y 367.423,Z 515.405,A -85,B 0,C 180,E1 13336.929,E2 13336.929} C_VEL
LIN {X 0,Y 363.999,Z 510.361,A -85,B 0,C 180,E1 13334.638,E2 13334.638} C_VEL
LIN {X 0,Y 361.091,Z 505.956,A -85,B 0,C 180,E1 13332.311,E2 13332.311} C_VEL
LIN {X 0,Y 358.287,Z 501.617,A -85,B 0,C 180,E1 13329.477,E2 13329.477} C_VEL
LIN {X 0,Y 355.241,Z 497.278,A -85,B 0,C 180,E1 13324.682,E2 13324.682} C_VEL
LIN {X 0,Y 354.877,Z 495.925,A -85,B 0,C 180,E1 13323.392,E2 13323.392} C_VEL
LIN {X 0,Y 354.947,Z 496.04,A -85,B 0,C 180,E1 13316.852,E2 13316.852} C_VEL
LIN {X 0,Y 356.737,Z 500.117,A -85,B 0,C 180,E1 13312.916,E2 13312.916} C_VEL
LIN {X 0,Y 358.408,Z 501.917,A -85,B 0,C 180,E1 13310.851,E2 13310.851} C_VEL
LIN {X 0,Y 361.264,Z 506.224,A -85,B 0,C 180,E1 13308.02,E2 13308.02} C_VEL
LIN {X 0,Y 365.408,Z 512.491,A -85,B 0,C 180,E1 13304.852,E2 13304.852} C_VEL
LIN {X 0,Y 368.961,Z 517.907,A -85,B 0,C 180,E1 13302.617,E2 13302.617} C_VEL
LIN {X 0,Y 372.88,Z 524.183,A -85,B 0,C 180,E1 13300.458,E2 13300.458} C_VEL
LIN {X 0,Y 378.215,Z 534.314,A -85,B 0,C 180,E1 13297.822,E2 13297.822} C_VEL
LIN {X 0,Y 362.932,Z 728.913,A -85,B 0,C 180,E1 13293.996,E2 13293.996} C_VEL
LIN {X 0,Y 359.478,Z 754.118,A -85,B 0,C 180,E1 13293.366,E2 13293.366} C_VEL
LIN {X 0,Y 355.042,Z 776.783,A -85,B 0,C 180,E1 13292.619,E2 13292.619} C_VEL
LIN {X 0,Y 349.424,Z 799.13,A -85,B 0,C 180,E1 13291.618,E2 13291.618} C_VEL
LIN {X 0,Y 343.159,Z 820.316,A -85,B 0,C 180,E1 13290.417,E2 13290.417} C_VEL
LIN {X 0,Y 336.054,Z 840.684,A -85,B 0,C 180,E1 13288.958,E2 13288.958} C_VEL
LIN {X 0,Y 327.918,Z 861.461,A -85,B 0,C 180,E1 13287.13,E2 13287.13} C_VEL
LIN {X 0,Y 320.158,Z 879.221,A -85,B 0,C 180,E1 13285.212,E2 13285.212} C_VEL
LIN {X 0,Y 310.79,Z 898.951,A -85,B 0,C 180,E1 13282.613,E2 13282.613} C_VEL
LIN {X 0,Y 302.464,Z 915.305,A -85,B 0,C 180,E1 13279.988,E2 13279.988} C_VEL
LIN {X 0,Y 293.608,Z 931.741,A -85,B 0,C 180,E1 13276.776,E2 13276.776} C_VEL
LIN {X 0,Y 285.272,Z 946.87,A -85,B 0,C 180,E1 13273.196,E2 13273.196} C_VEL
LIN {X 0,Y 277.734,Z 960.247,A -85,B 0,C 180,E1 13269.285,E2 13269.285} C_VEL
LIN {X 0,Y 270.948,Z 972.663,A -85,B 0,C 180,E1 13264.885,E2 13264.885} C_VEL
LIN {X 0,Y 265.715,Z 982.742,A -85,B 0,C 180,E1 13260.493,E2 13260.493} C_VEL
LIN {X 0,Y 261.294,Z 992.228,A -85,B 0,C 180,E1 13255.375,E2 13255.375} C_VEL
LIN {X 0,Y 258.57,Z 999.269,A -85,B 0,C 180,E1 13250.601,E2 13250.601} C_VEL
LIN {X 0,Y 256.873,Z 1004.939,A -85,B 0,C 180,E1 13245.578,E2 13245.578} C_VEL
LIN {X 0,Y 256.192,Z 1008.563,A -85,B 0,C 180,E1 13241.252,E2 13241.252} C_VEL
LIN {X 0,Y 255.987,Z 1011.268,A -85,B 0,C 180,E1 13236.504,E2 13236.504} C_VEL
LIN {X 0,Y 255.999,Z 1012.414,A -85,B 0,C 180,E1 13232.015,E2 13232.015} C_VEL
LIN {X 0,Y 256,Z 1012.437,A -85,B 0,C 180,E1 13228.21,E2 13228.21} C_VEL
LIN {X 0,Y 255.981,Z 1011.408,A -85,B 0,C 180,E1 13223.948,E2 13223.948} C_VEL
LIN {X 0,Y 256.149,Z 1008.887,A -85,B 0,C 180,E1 13219.203,E2 13219.203} C_VEL
LIN {X 0,Y 256.773,Z 1005.358,A -85,B 0,C 180,E1 13214.879,E2 13214.879} C_VEL
LIN {X 0,Y 258.367,Z 999.878,A -85,B 0,C 180,E1 13209.857,E2 13209.857} C_VEL
LIN {X 0,Y 261.137,Z 992.57,A -85,B 0,C 180,E1 13204.853,E2 13204.853} C_VEL
LIN {X 0,Y 265.294,Z 983.593,A -85,B 0,C 180,E1 13199.921,E2 13199.921} C_VEL
LIN {X 0,Y 270.37,Z 973.688,A -85,B 0,C 180,E1 13195.547,E2 13195.547} C_VEL
LIN {X 0,Y 277.404,Z 960.786,A -85,B 0,C 180,E1 13190.9,E2 13190.9} C_VEL
LIN {X 0,Y 284.711,Z 947.756,A -85,B 0,C 180,E1 13187.062,E2 13187.062} C_VEL
LIN {X 0,Y 292.649,Z 933.386,A -85,B 0,C 180,E1 13183.596,E2 13183.596} C_VEL
LIN {X 0,Y 301.305,Z 917.477,A -85,B 0,C 180,E1 13180.405,E2 13180.405} C_VEL
LIN {X 0,Y 309.932,Z 900.532,A -85,B 0,C 180,E1 13177.637,E2 13177.637} C_VEL
LIN {X 0,Y 318.722,Z 882.276,A -85,B 0,C 180,E1 13175.162,E2 13175.162} C_VEL
LIN {X 0,Y 326.952,Z 863.51,A -85,B 0,C 180,E1 13173.089,E2 13173.089} C_VEL
LIN {X 0,Y 335.37,Z 842.306,A -85,B 0,C 180,E1 13171.18,E2 13171.18} C_VEL
LIN {X 0,Y 342.101,Z 823.134,A -85,B 0,C 180,E1 13169.781,E2 13169.781} C_VEL
LIN {X 0,Y 348.696,Z 801.424,A -85,B 0,C 180,E1 13168.508,E2 13168.508} C_VEL
LIN {X 0,Y 354.203,Z 779.926,A -85,B 0,C 180,E1 13167.517,E2 13167.517} C_VEL
LIN {X 0,Y 358.921,Z 756.666,A -85,B 0,C 180,E1 13166.717,E2 13166.717} C_VEL
LIN {X 0,Y 362.403,Z 733.291,A -85,B 0,C 180,E1 13166.107,E2 13166.107} C_VEL
LIN {X 0,Y 367.726,Z 666.841,A -85,B 0,C 180,E1 13164.775,E2 13164.775} C_VEL
LIN {X 0,Y 378.106,Z 534.09,A -85,B 0,C 180,E1 13162.182,E2 13162.182} C_VEL
LIN {X 0,Y 372.12,Z 522.989,A -85,B 0,C 180,E1 13159.217,E2 13159.217} C_VEL
LIN {X 0,Y 367.268,Z 515.278,A -85,B 0,C 180,E1 13156.447,E2 13156.447} C_VEL
LIN {X 0,Y 363.725,Z 510.105,A -85,B 0,C 180,E1 13154.08,E2 13154.08} C_VEL
LIN {X 0,Y 361.096,Z 506.084,A -85,B 0,C 180,E1 13151.986,E2 13151.986} C_VEL
LIN {X 0,Y 358.297,Z 501.865,A -85,B 0,C 180,E1 13149.233,E2 13149.233} C_VEL
LIN {X 0,Y 355.106,Z 497.179,A -85,B 0,C 180,E1 13144.36,E2 13144.36} C_VEL
LIN {X 0,Y 354.707,Z 495.88,A -85,B 0,C 180,E1 13143.07,E2 13143.07} C_VEL
LIN {X 0,Y 354.792,Z 495.913,A -85,B 0,C 180,E1 13136.121,E2 13136.121} C_VEL
LIN {X 0,Y 356.951,Z 500.428,A -85,B 0,C 180,E1 13131.786,E2 13131.786} C_VEL
LIN {X 0,Y 358.295,Z 501.846,A -85,B 0,C 180,E1 13130.199,E2 13130.199} C_VEL
LIN {X 0,Y 361.835,Z 507.154,A -85,B 0,C 180,E1 13126.822,E2 13126.822} C_VEL
LIN {X 0,Y 365.37,Z 512.504,A -85,B 0,C 180,E1 13124.199,E2 13124.199} C_VEL
LIN {X 0,Y 369.272,Z 518.494,A -85,B 0,C 180,E1 13121.776,E2 13121.776} C_VEL
LIN {X 0,Y 375.123,Z 527.724,A -85,B 0,C 180,E1 13118.705,E2 13118.705} C_VEL
LIN {X 0,Y 377.983,Z 532.77,A -85,B 0,C 180,E1 13117.355,E2 13117.355} C_VEL
LIN {X 0,Y 363.26,Z 718.815,A -85,B 0,C 180,E1 13113.702,E2 13113.702} C_VEL
LIN {X 0,Y 359.95,Z 742.67,A -85,B 0,C 180,E1 13113.069,E2 13113.069} C_VEL
LIN {X 0,Y 356.063,Z 763.399,A -85,B 0,C 180,E1 13112.323,E2 13112.323} C_VEL
LIN {X 0,Y 350.947,Z 784.681,A -85,B 0,C 180,E1 13111.329,E2 13111.329} C_VEL
LIN {X 0,Y 345.53,Z 803.679,A -85,B 0,C 180,E1 13110.227,E2 13110.227} C_VEL
LIN {X 0,Y 338.494,Z 824.708,A -85,B 0,C 180,E1 13108.718,E2 13108.718} C_VEL
LIN {X 0,Y 331.542,Z 842.976,A -85,B 0,C 180,E1 13107.122,E2 13107.122} C_VEL
LIN {X 0,Y 323.222,Z 862.429,A -85,B 0,C 180,E1 13105.05,E2 13105.05} C_VEL
LIN {X 0,Y 315.04,Z 879.915,A -85,B 0,C 180,E1 13102.798,E2 13102.798} C_VEL
LIN {X 0,Y 306.23,Z 897.076,A -85,B 0,C 180,E1 13100.102,E2 13100.102} C_VEL
LIN {X 0,Y 297.608,Z 913.017,A -85,B 0,C 180,E1 13097.08,E2 13097.08} C_VEL
LIN {X 0,Y 289.314,Z 927.452,A -85,B 0,C 180,E1 13093.717,E2 13093.717} C_VEL
LIN {X 0,Y 281.187,Z 941.33,A -85,B 0,C 180,E1 13089.789,E2 13089.789} C_VEL
LIN {X 0,Y 274.579,Z 952.572,A -85,B 0,C 180,E1 13085.887,E2 13085.887} C_VEL
LIN {X 0,Y 268.279,Z 963.546,A -85,B 0,C 180,E1 13081.196,E2 13081.196} C_VEL
LIN {X 0,Y 263.445,Z 972.655,A -85,B 0,C 180,E1 13076.359,E2 13076.359} C_VEL
LIN {X 0,Y 259.983,Z 979.832,A -85,B 0,C 180,E1 13071.426,E2 13071.426} C_VEL
LIN {X 0,Y 257.767,Z 985.514,A -85,B 0,C 180,E1 13066.446,E2 13066.446} C_VEL
LIN {X 0,Y 256.618,Z 989.358,A -85,B 0,C 180,E1 13061.687,E2 13061.687} C_VEL
LIN {X 0,Y 256.144,Z 991.87,A -85,B 0,C 180,E1 13057.174,E2 13057.174} C_VEL
LIN {X 0,Y 256.01,Z 993.178,A -85,B 0,C 180,E1 13052.461,E2 13052.461} C_VEL
LIN {X 0,Y 256.007,Z 993.274,A -85,B 0,C 180,E1 13048.433,E2 13048.433} C_VEL
LIN {X 0,Y 256.082,Z 992.394,A -85,B 0,C 180,E1 13044.174,E2 13044.174} C_VEL
LIN {X 0,Y 256.466,Z 990.043,A -85,B 0,C 180,E1 13039.215,E2 13039.215} C_VEL
LIN {X 0,Y 257.402,Z 986.596,A -85,B 0,C 180,E1 13034.685,E2 13034.685} C_VEL
LIN {X 0,Y 259.45,Z 981.132,A -85,B 0,C 180,E1 13029.467,E2 13029.467} C_VEL
LIN {X 0,Y 262.472,Z 974.537,A -85,B 0,C 180,E1 13024.747,E2 13024.747} C_VEL
LIN {X 0,Y 267.214,Z 965.527,A -85,B 0,C 180,E1 13019.662,E2 13019.662} C_VEL
LIN {X 0,Y 272.614,Z 956.006,A -85,B 0,C 180,E1 13015.359,E2 13015.359} C_VEL
LIN {X 0,Y 279.587,Z 944.08,A -85,B 0,C 180,E1 13010.998,E2 13010.998} C_VEL
LIN {X 0,Y 287.058,Z 931.506,A -85,B 0,C 180,E1 13007.224,E2 13007.224} C_VEL
LIN {X 0,Y 295.072,Z 917.518,A -85,B 0,C 180,E1 13003.807,E2 13003.807} C_VEL
LIN {X 0,Y 303.583,Z 902.272,A -85,B 0,C 180,E1 13000.702,E2 13000.702} C_VEL
LIN {X 0,Y 310.954,Z 888.116,A -85,B 0,C 180,E1 12998.321,E2 12998.321} C_VEL
LIN {X 0,Y 313.035,Z 882.855,A -85,B 0,C 180,E1 12997.36,E2 12997.36} C_VEL
LIN {X 0,Y 316.252,Z 868.929,A -85,B 0,C 180,E1 12994.502,E2 12994.502} C_VEL
LIN {X 0,Y 318.176,Z 863.895,A -85,B 0,C 180,E1 12993.782,E2 12993.782} C_VEL
LIN {X 0,Y 326.403,Z 845.555,A -85,B 0,C 180,E1 12991.795,E2 12991.795} C_VEL
LIN {X 0,Y 333.968,Z 826.342,A -85,B 0,C 180,E1 12990.101,E2 12990.101} C_VEL
LIN {X 0,Y 341.108,Z 805.952,A -85,B 0,C 180,E1 12988.622,E2 12988.622} C_VEL
LIN {X 0,Y 347.036,Z 785.845,A -85,B 0,C 180,E1 12987.451,E2 12987.451} C_VEL
LIN {X 0,Y 352.486,Z 763.896,A -85,B 0,C 180,E1 12986.43,E2 12986.43} C_VEL
LIN {X 0,Y 356.495,Z 743.081,A -85,B 0,C 180,E1 12985.687,E2 12985.687} C_VEL
LIN {X 0,Y 359.89,Z 719.281,A -85,B 0,C 180,E1 12985.06,E2 12985.06} C_VEL
LIN {X 0,Y 374.673,Z 538.351,A -85,B 0,C 180,E1 12981.519,E2 12981.519} C_VEL
LIN {X 0,Y 374.698,Z 537.569,A -85,B 0,C 180,E1 12981.489,E2 12981.489} C_VEL
LIN {X 0,Y 369.541,Z 529.037,A -85,B 0,C 180,E1 12978.824,E2 12978.824} C_VEL
LIN {X 0,Y 365.108,Z 521.964,A -85,B 0,C 180,E1 12976.139,E2 12976.139} C_VEL
LIN {X 0,Y 362.487,Z 517.915,A -85,B 0,C 180,E1 12974.293,E2 12974.293} C_VEL
LIN {X 0,Y 359.753,Z 513.66,A -85,B 0,C 180,E1 12972.032,E2 12972.032} C_VEL
LIN {X 0,Y 356.76,Z 509.087,A -85,B 0,C 180,E1 12968.867,E2 12968.867} C_VEL
LIN {X 0,Y 354.148,Z 504.983,A -85,B 0,C 180,E1 12964.372,E2 12964.372} C_VEL
LIN {X 0,Y 353.852,Z 503.851,A -85,B 0,C 180,E1 12963.24,E2 12963.24} C_VEL
LIN {X 0,Y 353.903,Z 503.857,A -85,B 0,C 180,E1 12957.085,E2 12957.085} C_VEL
LIN {X 0,Y 355.651,Z 507.995,A -85,B 0,C 180,E1 12953.057,E2 12953.057} C_VEL
LIN {X 0,Y 357.216,Z 509.756,A -85,B 0,C 180,E1 12951.064,E2 12951.064} C_VEL
LIN {X 0,Y 360.105,Z 514.115,A -85,B 0,C 180,E1 12948.144,E2 12948.144} C_VEL
LIN {X 0,Y 363.965,Z 520.223,A -85,B 0,C 180,E1 12945.117,E2 12945.117} C_VEL
LIN {X 0,Y 367.262,Z 525.367,A -85,B 0,C 180,E1 12942.983,E2 12942.983} C_VEL
LIN {X 0,Y 371.226,Z 531.934,A -85,B 0,C 180,E1 12940.735,E2 12940.735} C_VEL
LIN {X 0,Y 374.817,Z 539.264,A -85,B 0,C 180,E1 12938.86,E2 12938.86} C_VEL
LIN {X 0,Y 359.37,Z 729.714,A -85,B 0,C 180,E1 12935.126,E2 12935.126} C_VEL
LIN {X 0,Y 355.866,Z 754.26,A -85,B 0,C 180,E1 12934.511,E2 12934.511} C_VEL
LIN {X 0,Y 351.336,Z 776.817,A -85,B 0,C 180,E1 12933.775,E2 12933.775} C_VEL
LIN {X 0,Y 345.489,Z 799.398,A -85,B 0,C 180,E1 12932.772,E2 12932.772} C_VEL
LIN {X 0,Y 338.86,Z 821.028,A -85,B 0,C 180,E1 12931.546,E2 12931.546} C_VEL
LIN {X 0,Y 331.572,Z 841.29,A -85,B 0,C 180,E1 12930.096,E2 12930.096} C_VEL
LIN {X 0,Y 322.883,Z 862.623,A -85,B 0,C 180,E1 12928.206,E2 12928.206} C_VEL
LIN {X 0,Y 314.599,Z 880.916,A -85,B 0,C 180,E1 12926.208,E2 12926.208} C_VEL
LIN {X 0,Y 305.236,Z 899.767,A -85,B 0,C 180,E1 12923.681,E2 12923.681} C_VEL
LIN {X 0,Y 296.251,Z 916.758,A -85,B 0,C 180,E1 12920.912,E2 12920.912} C_VEL
LIN {X 0,Y 287.456,Z 932.288,A -85,B 0,C 180,E1 12917.8,E2 12917.8} C_VEL
LIN {X 0,Y 279.078,Z 946.785,A -85,B 0,C 180,E1 12914.312,E2 12914.312} C_VEL
LIN {X 0,Y 271.325,Z 959.869,A -85,B 0,C 180,E1 12910.43,E2 12910.43} C_VEL
LIN {X 0,Y 264.004,Z 972.515,A -85,B 0,C 180,E1 12905.858,E2 12905.858} C_VEL
LIN {X 0,Y 258.569,Z 982.366,A -85,B 0,C 180,E1 12901.465,E2 12901.465} C_VEL
LIN {X 0,Y 253.791,Z 991.916,A -85,B 0,C 180,E1 12896.181,E2 12896.181} C_VEL
LIN {X 0,Y 250.84,Z 998.96,A -85,B 0,C 180,E1 12891.266,E2 12891.266} C_VEL
LIN {X 0,Y 248.985,Z 1004.632,A -85,B 0,C 180,E1 12886.085,E2 12886.085} C_VEL
LIN {X 0,Y 248.225,Z 1008.259,A -85,B 0,C 180,E1 12881.618,E2 12881.618} C_VEL
LIN {X 0,Y 247.985,Z 1010.966,A -85,B 0,C 180,E1 12876.715,E2 12876.715} C_VEL
LIN {X 0,Y 248.002,Z 1012.114,A -85,B 0,C 180,E1 12872.08,E2 12872.08} C_VEL
LIN {X 0,Y 248.005,Z 1012.137,A -85,B 0,C 180,E1 12868.153,E2 12868.153} C_VEL
LIN {X 0,Y 247.99,Z 1011.107,A -85,B 0,C 180,E1 12863.752,E2 12863.752} C_VEL
LIN {X 0,Y 248.181,Z 1008.582,A -85,B 0,C 180,E1 12858.852,E2 12858.852} C_VEL
LIN {X 0,Y 248.87,Z 1005.05,A -85,B 0,C 180,E1 12854.387,E2 12854.387} C_VEL
LIN {X 0,Y 250.622,Z 999.567,A -85,B 0,C 180,E1 12849.206,E2 12849.206} C_VEL
LIN {X 0,Y 253.619,Z 992.256,A -85,B 0,C 180,E1 12844.053,E2 12844.053} C_VEL
LIN {X 0,Y 258.25,Z 982.945,A -85,B 0,C 180,E1 12838.829,E2 12838.829} C_VEL
LIN {X 0,Y 263.788,Z 972.844,A -85,B 0,C 180,E1 12834.293,E2 12834.293} C_VEL
LIN {X 0,Y 270.942,Z 960.469,A -85,B 0,C 180,E1 12829.78,E2 12829.78} C_VEL
LIN {X 0,Y 278.724,Z 947.285,A -85,B 0,C 180,E1 12825.844,E2 12825.844} C_VEL
LIN {X 0,Y 286.949,Z 933.07,A -85,B 0,C 180,E1 12822.387,E2 12822.387} C_VEL
LIN {X 0,Y 295.957,Z 917.181,A -85,B 0,C 180,E1 12819.179,E2 12819.179} C_VEL
LIN {X 0,Y 304.901,Z 900.271,A -85,B 0,C 180,E1 12816.409,E2 12816.409} C_VEL
LIN {X 0,Y 314.261,Z 881.468,A -85,B 0,C 180,E1 12813.871,E2 12813.871} C_VEL
LIN {X 0,Y 322.537,Z 863.198,A -85,B 0,C 180,E1 12811.866,E2 12811.866} C_VEL
LIN {X 0,Y 331.211,Z 841.994,A -85,B 0,C 180,E1 12809.97,E2 12809.97} C_VEL
LIN {X 0,Y 338.13,Z 822.822,A -85,B 0,C 180,E1 12808.583,E2 12808.583} C_VEL
LIN {X 0,Y 344.901,Z 801.112,A -85,B 0,C 180,E1 12807.324,E2 12807.324} C_VEL
LIN {X 0,Y 350.568,Z 779.515,A -85,B 0,C 180,E1 12806.342,E2 12806.342} C_VEL
LIN {X 0,Y 355.374,Z 756.352,A -85,B 0,C 180,E1 12805.557,E2 12805.557} C_VEL
LIN {X 0,Y 358.934,Z 732.969,A -85,B 0,C 180,E1 12804.953,E2 12804.953} C_VEL
LIN {X 0,Y 364.445,Z 666.259,A -85,B 0,C 180,E1 12803.62,E2 12803.62} C_VEL
LIN {X 0,Y 374.666,Z 538.791,A -85,B 0,C 180,E1 12801.116,E2 12801.116} C_VEL
LIN {X 0,Y 369.861,Z 529.7,A -85,B 0,C 180,E1 12798.602,E2 12798.602} C_VEL
LIN {X 0,Y 365.423,Z 522.501,A -85,B 0,C 180,E1 12795.961,E2 12795.961} C_VEL
LIN {X 0,Y 362.213,Z 517.654,A -85,B 0,C 180,E1 12793.732,E2 12793.732} C_VEL
LIN {X 0,Y 359.75,Z 513.787,A -85,B 0,C 180,E1 12791.706,E2 12791.706} C_VEL
LIN {X 0,Y 356.977,Z 509.409,A -85,B 0,C 180,E1 12788.861,E2 12788.861} C_VEL
LIN {X 0,Y 354.115,Z 505.268,A -85,B 0,C 180,E1 12784.372,E2 12784.372} C_VEL
LIN {X 0,Y 353.733,Z 503.822,A -85,B 0,C 180,E1 12783.078,E2 12783.078} C_VEL
LIN {X 0,Y 353.788,Z 503.856,A -85,B 0,C 180,E1 12776.192,E2 12776.192} C_VEL
LIN {X 0,Y 355.624,Z 508.037,A -85,B 0,C 180,E1 12772.244,E2 12772.244} C_VEL
LIN {X 0,Y 357.101,Z 509.685,A -85,B 0,C 180,E1 12770.41,E2 12770.41} C_VEL
LIN {X 0,Y 360.47,Z 514.87,A -85,B 0,C 180,E1 12767.097,E2 12767.097} C_VEL
LIN {X 0,Y 363.816,Z 520.056,A -85,B 0,C 180,E1 12764.539,E2 12764.539} C_VEL
LIN {X 0,Y 368.413,Z 527.18,A -85,B 0,C 180,E1 12761.65,E2 12761.65} C_VEL
LIN {X 0,Y 374.249,Z 536.938,A -85,B 0,C 180,E1 12758.571,E2 12758.571} C_VEL
LIN {X 0,Y 374.591,Z 537.754,A -85,B 0,C 180,E1 12758.394,E2 12758.394} C_VEL
LIN {X 0,Y 359.77,Z 719.313,A -85,B 0,C 180,E1 12754.84,E2 12754.84} C_VEL
LIN {X 0,Y 356.373,Z 743.114,A -85,B 0,C 180,E1 12754.213,E2 12754.213} C_VEL
LIN {X 0,Y 352.365,Z 763.927,A -85,B 0,C 180,E1 12753.469,E2 12753.469} C_VEL
LIN {X 0,Y 347.162,Z 784.991,A -85,B 0,C 180,E1 12752.493,E2 12752.493} C_VEL
LIN {X 0,Y 341.597,Z 803.989,A -85,B 0,C 180,E1 12751.401,E2 12751.401} C_VEL
LIN {X 0,Y 334.455,Z 824.772,A -85,B 0,C 180,E1 12749.923,E2 12749.923} C_VEL
LIN {X 0,Y 327.196,Z 843.308,A -85,B 0,C 180,E1 12748.314,E2 12748.314} C_VEL
LIN {X 0,Y 318.624,Z 862.739,A -85,B 0,C 180,E1 12746.251,E2 12746.251} C_VEL
LIN {X 0,Y 309.873,Z 880.826,A -85,B 0,C 180,E1 12743.918,E2 12743.918} C_VEL
LIN {X 0,Y 300.759,Z 897.887,A -85,B 0,C 180,E1 12741.213,E2 12741.213} C_VEL
LIN {X 0,Y 292.064,Z 913.329,A -85,B 0,C 180,E1 12738.263,E2 12738.263} C_VEL
LIN {X 0,Y 283.402,Z 927.764,A -85,B 0,C 180,E1 12734.872,E2 12734.872} C_VEL
LIN {X 0,Y 274.678,Z 941.966,A -85,B 0,C 180,E1 12730.786,E2 12730.786} C_VEL
LIN {X 0,Y 267.58,Z 953.445,A -85,B 0,C 180,E1 12726.712,E2 12726.712} C_VEL
LIN {X 0,Y 261.235,Z 963.858,A -85,B 0,C 180,E1 12722.137,E2 12722.137} C_VEL
LIN {X 0,Y 256.078,Z 972.965,A -85,B 0,C 180,E1 12717.178,E2 12717.178} C_VEL
LIN {X 0,Y 252.358,Z 980.141,A -85,B 0,C 180,E1 12712.107,E2 12712.107} C_VEL
LIN {X 0,Y 249.955,Z 985.82,A -85,B 0,C 180,E1 12706.976,E2 12706.976} C_VEL
LIN {X 0,Y 248.694,Z 989.662,A -85,B 0,C 180,E1 12702.065,E2 12702.065} C_VEL
LIN {X 0,Y 248.162,Z 992.173,A -85,B 0,C 180,E1 12697.406,E2 12697.406} C_VEL
LIN {X 0,Y 248.015,Z 993.478,A -85,B 0,C 180,E1 12692.541,E2 12692.541} C_VEL
LIN {X 0,Y 248.013,Z 993.573,A -85,B 0,C 180,E1 12688.382,E2 12688.382} C_VEL
LIN {X 0,Y 248.098,Z 992.695,A -85,B 0,C 180,E1 12683.985,E2 12683.985} C_VEL
LIN {X 0,Y 248.5,Z 990.461,A -85,B 0,C 180,E1 12679.04,E2 12679.04} C_VEL
LIN {X 0,Y 249.547,Z 986.901,A -85,B 0,C 180,E1 12674.191,E2 12674.191} C_VEL
LIN {X 0,Y 251.683,Z 981.676,A -85,B 0,C 180,E1 12669.001,E2 12669.001} C_VEL
LIN {X 0,Y 254.856,Z 975.188,A -85,B 0,C 180,E1 12664.187,E2 12664.187} C_VEL
LIN {X 0,Y 259.608,Z 966.73,A -85,B 0,C 180,E1 12659.19,E2 12659.19} C_VEL
LIN {X 0,Y 265.527,Z 956.817,A -85,B 0,C 180,E1 12654.561,E2 12654.561} C_VEL
LIN {X 0,Y 272.821,Z 945.011,A -85,B 0,C 180,E1 12650.112,E2 12650.112} C_VEL
LIN {X 0,Y 280.607,Z 932.501,A -85,B 0,C 180,E1 12646.276,E2 12646.276} C_VEL
LIN {X 0,Y 288.936,Z 918.656,A -85,B 0,C 180,E1 12642.815,E2 12642.815} C_VEL
LIN {X 0,Y 297.966,Z 903.152,A -85,B 0,C 180,E1 12639.611,E2 12639.611} C_VEL
LIN {X 0,Y 307.078,Z 886.249,A -85,B 0,C 180,E1 12636.784,E2 12636.784} C_VEL
LIN {X 0,Y 316.014,Z 868.543,A -85,B 0,C 180,E1 12634.34,E2 12634.34} C_VEL
LIN {X 0,Y 318.176,Z 863.895,A -85,B 0,C 180,E1 12633.782,E2 12633.782} C_VEL
LIN {X 0,Y 320.359,Z 858.127,A -85,B 0,C 180,E1 12632.948,E2 12632.948} C_VEL
LIN {X 0,Y 323.649,Z 843.632,A -85,B 0,C 180,E1 12630.525,E2 12630.525} C_VEL
LIN {X 0,Y 325.692,Z 837.437,A -85,B 0,C 180,E1 12629.789,E2 12629.789} C_VEL
LIN {X 0,Y 333.786,Z 816.359,A -85,B 0,C 180,E1 12628.105,E2 12628.105} C_VEL
LIN {X 0,Y 340.5,Z 796.143,A -85,B 0,C 180,E1 12626.8,E2 12626.8} C_VEL
LIN {X 0,Y 346.613,Z 773.936,A -85,B 0,C 180,E1 12625.663,E2 12625.663} C_VEL
LIN {X 0,Y 351.693,Z 751.284,A -85,B 0,C 180,E1 12624.762,E2 12624.762} C_VEL
LIN {X 0,Y 355.435,Z 728.365,A -85,B 0,C 180,E1 12624.1,E2 12624.1} C_VEL
LIN {X 0,Y 358.402,Z 699.941,A -85,B 0,C 180,E1 12623.493,E2 12623.493} C_VEL
LIN {X 0,Y 371.459,Z 542.597,A -85,B 0,C 180,E1 12620.442,E2 12620.442} C_VEL
LIN {X 0,Y 366.024,Z 533.537,A -85,B 0,C 180,E1 12617.405,E2 12617.405} C_VEL
LIN {X 0,Y 361.615,Z 526.271,A -85,B 0,C 180,E1 12614.41,E2 12614.41} C_VEL
LIN {X 0,Y 358.424,Z 521.363,A -85,B 0,C 180,E1 12611.75,E2 12611.75} C_VEL
LIN {X 0,Y 355.655,Z 516.967,A -85,B 0,C 180,E1 12608.732,E2 12608.732} C_VEL
LIN {X 0,Y 353.111,Z 512.878,A -85,B 0,C 180,E1 12604.222,E2 12604.222} C_VEL
LIN {X 0,Y 352.829,Z 511.778,A -85,B 0,C 180,E1 12603.087,E2 12603.087} C_VEL
LIN {X 0,Y 352.913,Z 511.933,A -85,B 0,C 180,E1 12597.077,E2 12597.077} C_VEL
LIN {X 0,Y 354.676,Z 515.995,A -85,B 0,C 180,E1 12593.038,E2 12593.038} C_VEL
LIN {X 0,Y 356.029,Z 517.59,A -85,B 0,C 180,E1 12591.278,E2 12591.278} C_VEL
LIN {X 0,Y 359.279,Z 522.747,A -85,B 0,C 180,E1 12587.953,E2 12587.953} C_VEL
LIN {X 0,Y 362.53,Z 527.952,A -85,B 0,C 180,E1 12585.383,E2 12585.383} C_VEL
LIN {X 0,Y 365.885,Z 533.316,A -85,B 0,C 180,E1 12583.162,E2 12583.162} C_VEL
LIN {X 0,Y 369.638,Z 539.906,A -85,B 0,C 180,E1 12580.977,E2 12580.977} C_VEL
LIN {X 0,Y 371.56,Z 544.032,A -85,B 0,C 180,E1 12579.92,E2 12579.92} C_VEL
LIN {X 0,Y 356.001,Z 730.021,A -85,B 0,C 180,E1 12576.288,E2 12576.288} C_VEL
LIN {X 0,Y 352.432,Z 754.222,A -85,B 0,C 180,E1 12575.685,E2 12575.685} C_VEL
LIN {X 0,Y 347.866,Z 776.438,A -85,B 0,C 180,E1 12574.97,E2 12574.97} C_VEL
LIN {X 0,Y 342.131,Z 798.169,A -85,B 0,C 180,E1 12574.024,E2 12574.024} C_VEL
LIN {X 0,Y 335.43,Z 819.718,A -85,B 0,C 180,E1 12572.833,E2 12572.833} C_VEL
LIN {X 0,Y 327.89,Z 840.184,A -85,B 0,C 180,E1 12571.397,E2 12571.397} C_VEL
LIN {X 0,Y 319.32,Z 860.827,A -85,B 0,C 180,E1 12569.608,E2 12569.608} C_VEL
LIN {X 0,Y 310.719,Z 879.285,A -85,B 0,C 180,E1 12567.63,E2 12567.63} C_VEL
LIN {X 0,Y 300.699,Z 898.897,A -85,B 0,C 180,E1 12565.04,E2 12565.04} C_VEL
LIN {X 0,Y 291.343,Z 915.936,A -85,B 0,C 180,E1 12562.276,E2 12562.276} C_VEL
LIN {X 0,Y 281.909,Z 931.978,A -85,B 0,C 180,E1 12559.058,E2 12559.058} C_VEL
LIN {X 0,Y 273.145,Z 946.473,A -85,B 0,C 180,E1 12555.539,E2 12555.539} C_VEL
LIN {X 0,Y 264.983,Z 959.556,A -85,B 0,C 180,E1 12551.608,E2 12551.608} C_VEL
LIN {X 0,Y 257.348,Z 972.036,A -85,B 0,C 180,E1 12547.024,E2 12547.024} C_VEL
LIN {X 0,Y 251.46,Z 982.053,A -85,B 0,C 180,E1 12542.462,E2 12542.462} C_VEL
LIN {X 0,Y 246.34,Z 991.605,A -85,B 0,C 180,E1 12537.036,E2 12537.036} C_VEL
LIN {X 0,Y 243.137,Z 998.65,A -85,B 0,C 180,E1 12531.974,E2 12531.974} C_VEL
LIN {X 0,Y 241.114,Z 1004.325,A -85,B 0,C 180,E1 12526.625,E2 12526.625} C_VEL
LIN {X 0,Y 240.261,Z 1007.954,A -85,B 0,C 180,E1 12522.009,E2 12522.009} C_VEL
LIN {X 0,Y 239.982,Z 1010.664,A -85,B 0,C 180,E1 12516.94,E2 12516.94} C_VEL
LIN {X 0,Y 239.999,Z 1011.79,A -85,B 0,C 180,E1 12512.388,E2 12512.388} C_VEL
LIN {X 0,Y 240.011,Z 1011.861,A -85,B 0,C 180,E1 12508.33,E2 12508.33} C_VEL
LIN {X 0,Y 239.987,Z 1010.949,A -85,B 0,C 180,E1 12504.023,E2 12504.023} C_VEL
LIN {X 0,Y 240.169,Z 1008.609,A -85,B 0,C 180,E1 12498.961,E2 12498.961} C_VEL
LIN {X 0,Y 240.923,Z 1004.957,A -85,B 0,C 180,E1 12494.106,E2 12494.106} C_VEL
LIN {X 0,Y 242.675,Z 999.808,A -85,B 0,C 180,E1 12488.998,E2 12488.998} C_VEL
LIN {X 0,Y 245.793,Z 992.671,A -85,B 0,C 180,E1 12483.683,E2 12483.683} C_VEL
LIN {X 0,Y 250.443,Z 983.902,A -85,B 0,C 180,E1 12478.471,E2 12478.471} C_VEL
LIN {X 0,Y 256.373,Z 973.582,A -85,B 0,C 180,E1 12473.65,E2 12473.65} C_VEL
LIN {X 0,Y 263.806,Z 961.449,A -85,B 0,C 180,E1 12469.034,E2 12469.034} C_VEL
LIN {X 0,Y 271.312,Z 949.265,A -85,B 0,C 180,E1 12465.268,E2 12465.268} C_VEL
LIN {X 0,Y 280.874,Z 933.613,A -85,B 0,C 180,E1 12461.321,E2 12461.321} C_VEL
LIN {X 0,Y 289.932,Z 918.259,A -85,B 0,C 180,E1 12458.17,E2 12458.17} C_VEL
LIN {X 0,Y 299.565,Z 900.862,A -85,B 0,C 180,E1 12455.269,E2 12455.269} C_VEL
LIN {X 0,Y 309.099,Z 882.504,A -85,B 0,C 180,E1 12452.762,E2 12452.762} C_VEL
LIN {X 0,Y 317.938,Z 863.627,A -85,B 0,C 180,E1 12450.684,E2 12450.684} C_VEL
LIN {X 0,Y 326.856,Z 842.589,A -85,B 0,C 180,E1 12448.801,E2 12448.801} C_VEL
LIN {X 0,Y 333.913,Z 823.623,A -85,B 0,C 180,E1 12447.431,E2 12447.431} C_VEL
LIN {X 0,Y 341.258,Z 800.801,A -85,B 0,C 180,E1 12446.116,E2 12446.116} C_VEL
LIN {X 0,Y 346.869,Z 779.946,A -85,B 0,C 180,E1 12445.177,E2 12445.177} C_VEL
LIN {X 0,Y 351.904,Z 756.429,A -85,B 0,C 180,E1 12444.386,E2 12444.386} C_VEL
LIN {X 0,Y 355.58,Z 732.966,A -85,B 0,C 180,E1 12443.784,E2 12443.784} C_VEL
LIN {X 0,Y 360.949,Z 670.145,A -85,B 0,C 180,E1 12442.532,E2 12442.532} C_VEL
LIN {X 0,Y 371.434,Z 543.659,A -85,B 0,C 180,E1 12440.072,E2 12440.072} C_VEL
LIN {X 0,Y 367.647,Z 536.398,A -85,B 0,C 180,E1 12437.979,E2 12437.979} C_VEL
LIN {X 0,Y 363.489,Z 529.549,A -85,B 0,C 180,E1 12435.393,E2 12435.393} C_VEL
LIN {X 0,Y 360.714,Z 525.202,A -85,B 0,C 180,E1 12433.382,E2 12433.382} C_VEL
LIN {X 0,Y 358.413,Z 521.49,A -85,B 0,C 180,E1 12431.424,E2 12431.424} C_VEL
LIN {X 0,Y 355.458,Z 516.855,A -85,B 0,C 180,E1 12428.248,E2 12428.248} C_VEL
LIN {X 0,Y 353.015,Z 512.97,A -85,B 0,C 180,E1 12424.06,E2 12424.06} C_VEL
LIN {X 0,Y 352.705,Z 511.743,A -85,B 0,C 180,E1 12422.925,E2 12422.925} C_VEL
LIN {X 0,Y 352.758,Z 511.772,A -85,B 0,C 180,E1 12416.343,E2 12416.343} C_VEL
LIN {X 0,Y 354.649,Z 516.052,A -85,B 0,C 180,E1 12412.222,E2 12412.222} C_VEL
LIN {X 0,Y 355.913,Z 517.52,A -85,B 0,C 180,E1 12410.622,E2 12410.622} C_VEL
LIN {X 0,Y 359.115,Z 522.583,A -85,B 0,C 180,E1 12407.375,E2 12407.375} C_VEL
LIN {X 0,Y 362.274,Z 527.608,A -85,B 0,C 180,E1 12404.881,E2 12404.881} C_VEL
LIN {X 0,Y 366.632,Z 534.56,A -85,B 0,C 180,E1 12402.051,E2 12402.051} C_VEL
LIN {X 0,Y 371.337,Z 542.593,A -85,B 0,C 180,E1 12399.453,E2 12399.453} C_VEL
LIN {X 0,Y 356.442,Z 719.633,A -85,B 0,C 180,E1 12396.004,E2 12396.004} C_VEL
LIN {X 0,Y 352.964,Z 743.427,A -85,B 0,C 180,E1 12395.383,E2 12395.383} C_VEL
LIN {X 0,Y 348.879,Z 764.131,A -85,B 0,C 180,E1 12394.652,E2 12394.652} C_VEL
LIN {X 0,Y 343.523,Z 785.301,A -85,B 0,C 180,E1 12393.683,E2 12393.683} C_VEL
LIN {X 0,Y 337.463,Z 805.421,A -85,B 0,C 180,E1 12392.532,E2 12392.532} C_VEL
LIN {X 0,Y 330.131,Z 825.974,A -85,B 0,C 180,E1 12391.066,E2 12391.066} C_VEL
LIN {X 0,Y 322.348,Z 845.223,A -85,B 0,C 180,E1 12389.389,E2 12389.389} C_VEL
LIN {X 0,Y 313.975,Z 863.449,A -85,B 0,C 180,E1 12387.44,E2 12387.44} C_VEL
LIN {X 0,Y 305.129,Z 881.137,A -85,B 0,C 180,E1 12385.159,E2 12385.159} C_VEL
LIN {X 0,Y 295.977,Z 897.698,A -85,B 0,C 180,E1 12382.539,E2 12382.539} C_VEL
LIN {X 0,Y 286.652,Z 913.64,A -85,B 0,C 180,E1 12379.49,E2 12379.49} C_VEL
LIN {X 0,Y 277.611,Z 928.077,A -85,B 0,C 180,E1 12376.074,E2 12376.074} C_VEL
LIN {X 0,Y 268.692,Z 941.955,A -85,B 0,C 180,E1 12372.046,E2 12372.046} C_VEL
LIN {X 0,Y 261.25,Z 953.337,A -85,B 0,C 180,E1 12367.963,E2 12367.963} C_VEL
LIN {X 0,Y 254.234,Z 964.222,A -85,B 0,C 180,E1 12363.102,E2 12363.102} C_VEL
LIN {X 0,Y 248.767,Z 973.276,A -85,B 0,C 180,E1 12358.046,E2 12358.046} C_VEL
LIN {X 0,Y 244.767,Z 980.45,A -85,B 0,C 180,E1 12352.831,E2 12352.831} C_VEL
LIN {X 0,Y 242.138,Z 986.184,A -85,B 0,C 180,E1 12347.47,E2 12347.47} C_VEL
LIN {X 0,Y 240.774,Z 989.967,A -85,B 0,C 180,E1 12342.469,E2 12342.469} C_VEL
LIN {X 0,Y 240.186,Z 992.475,A -85,B 0,C 180,E1 12337.654,E2 12337.654} C_VEL
LIN {X 0,Y 240.02,Z 993.778,A -85,B 0,C 180,E1 12332.625,E2 12332.625} C_VEL
LIN {X 0,Y 240.02,Z 993.873,A -85,B 0,C 180,E1 12328.329,E2 12328.329} C_VEL
LIN {X 0,Y 240.115,Z 992.996,A -85,B 0,C 180,E1 12323.785,E2 12323.785} C_VEL
LIN {X 0,Y 240.553,Z 990.803,A -85,B 0,C 180,E1 12318.735,E2 12318.735} C_VEL
LIN {X 0,Y 241.636,Z 987.405,A -85,B 0,C 180,E1 12313.906,E2 12313.906} C_VEL
LIN {X 0,Y 243.935,Z 982.22,A -85,B 0,C 180,E1 12308.505,E2 12308.505} C_VEL
LIN {X 0,Y 247.46,Z 975.495,A -85,B 0,C 180,E1 12303.356,E2 12303.356} C_VEL
LIN {X 0,Y 252.539,Z 967.039,A -85,B 0,C 180,E1 12298.229,E2 12298.229} C_VEL
LIN {X 0,Y 258.492,Z 957.628,A -85,B 0,C 180,E1 12293.719,E2 12293.719} C_VEL
LIN {X 0,Y 266.618,Z 945.169,A -85,B 0,C 180,E1 12288.92,E2 12288.92} C_VEL
LIN {X 0,Y 275.158,Z 932.121,A -85,B 0,C 180,E1 12284.886,E2 12284.886} C_VEL
LIN {X 0,Y 283.903,Z 918.131,A -85,B 0,C 180,E1 12281.403,E2 12281.403} C_VEL
LIN {X 0,Y 293.293,Z 902.589,A -85,B 0,C 180,E1 12278.213,E2 12278.213} C_VEL
LIN {X 0,Y 302.451,Z 886.187,A -85,B 0,C 180,E1 12275.486,E2 12275.486} C_VEL
LIN {X 0,Y 312.119,Z 867.523,A -85,B 0,C 180,E1 12272.943,E2 12272.943} C_VEL
LIN {X 0,Y 320.207,Z 850.244,A -85,B 0,C 180,E1 12271.012,E2 12271.012} C_VEL
LIN {X 0,Y 325.692,Z 837.437,A -85,B 0,C 180,E1 12269.789,E2 12269.789} C_VEL
LIN {X 0,Y 327.807,Z 831.142,A -85,B 0,C 180,E1 12269.088,E2 12269.088} C_VEL
LIN {X 0,Y 330.943,Z 815.501,A -85,B 0,C 180,E1 12266.955,E2 12266.955} C_VEL
LIN {X 0,Y 332.877,Z 808.899,A -85,B 0,C 180,E1 12266.342,E2 12266.342} C_VEL
LIN {X 0,Y 339.56,Z 787.68,A -85,B 0,C 180,E1 12265.109,E2 12265.109} C_VEL
LIN {X 0,Y 345.105,Z 766.865,A -85,B 0,C 180,E1 12264.141,E2 12264.141} C_VEL
LIN {X 0,Y 349.613,Z 744.952,A -85,B 0,C 180,E1 12263.362,E2 12263.362} C_VEL
LIN {X 0,Y 353.208,Z 721.758,A -85,B 0,C 180,E1 12262.749,E2 12262.749} C_VEL
LIN {X 0,Y 359.599,Z 649.033,A -85,B 0,C 180,E1 12261.318,E2 12261.318} C_VEL
LIN {X 0,Y 368.259,Z 547.736,A -85,B 0,C 180,E1 12259.344,E2 12259.344} C_VEL
LIN {X 0,Y 363.513,Z 539.614,A -85,B 0,C 180,E1 12256.499,E2 12256.499} C_VEL
LIN {X 0,Y 359.602,Z 533.159,A -85,B 0,C 180,E1 12253.671,E2 12253.671} C_VEL
LIN {X 0,Y 357.103,Z 529.065,A -85,B 0,C 180,E1 12251.467,E2 12251.467} C_VEL
LIN {X 0,Y 354.421,Z 524.74,A -85,B 0,C 180,E1 12248.436,E2 12248.436} C_VEL
LIN {X 0,Y 352.034,Z 520.583,A -85,B 0,C 180,E1 12243.909,E2 12243.909} C_VEL
LIN {X 0,Y 351.809,Z 519.706,A -85,B 0,C 180,E1 12242.933,E2 12242.933} C_VEL
LIN {X 0,Y 351.891,Z 519.828,A -85,B 0,C 180,E1 12237.232,E2 12237.232} C_VEL
LIN {X 0,Y 353.591,Z 523.873,A -85,B 0,C 180,E1 12233.18,E2 12233.18} C_VEL
LIN {X 0,Y 354.847,Z 525.423,A -85,B 0,C 180,E1 12231.493,E2 12231.493} C_VEL
LIN {X 0,Y 357.932,Z 530.454,A -85,B 0,C 180,E1 12228.234,E2 12228.234} C_VEL
LIN {X 0,Y 361.103,Z 535.677,A -85,B 0,C 180,E1 12225.652,E2 12225.652} C_VEL
LIN {X 0,Y 364.948,Z 541.919,A -85,B 0,C 180,E1 12223.077,E2 12223.077} C_VEL
LIN {X 0,Y 368.437,Z 548.649,A -85,B 0,C 180,E1 12221.006,E2 12221.006} C_VEL
LIN {X 0,Y 352.835,Z 729.813,A -85,B 0,C 180,E1 12217.483,E2 12217.483} C_VEL
LIN {X 0,Y 349.18,Z 754.017,A -85,B 0,C 180,E1 12216.886,E2 12216.886} C_VEL
LIN {X 0,Y 344.586,Z 775.907,A -85,B 0,C 180,E1 12216.193,E2 12216.193} C_VEL
LIN {X 0,Y 338.517,Z 798.373,A -85,B 0,C 180,E1 12215.231,E2 12215.231} C_VEL
LIN {X 0,Y 331.666,Z 819.777,A -85,B 0,C 180,E1 12214.059,E2 12214.059} C_VEL
LIN {X 0,Y 324.102,Z 839.782,A -85,B 0,C 180,E1 12212.672,E2 12212.672} C_VEL
LIN {X 0,Y 315.595,Z 859.794,A -85,B 0,C 180,E1 12210.965,E2 12210.965} C_VEL
LIN {X 0,Y 306.64,Z 878.467,A -85,B 0,C 180,E1 12208.991,E2 12208.991} C_VEL
LIN {X 0,Y 296.344,Z 898.028,A -85,B 0,C 180,E1 12206.438,E2 12206.438} C_VEL
LIN {X 0,Y 286.905,Z 914.599,A -85,B 0,C 180,E1 12203.774,E2 12203.774} C_VEL
LIN {X 0,Y 277.036,Z 930.808,A -85,B 0,C 180,E1 12200.559,E2 12200.559} C_VEL
LIN {X 0,Y 267.831,Z 945.414,A -85,B 0,C 180,E1 12197.023,E2 12197.023} C_VEL
LIN {X 0,Y 259.183,Z 958.595,A -85,B 0,C 180,E1 12193.059,E2 12193.059} C_VEL
LIN {X 0,Y 251.411,Z 970.668,A -85,B 0,C 180,E1 12188.633,E2 12188.633} C_VEL
LIN {X 0,Y 244.708,Z 981.269,A -85,B 0,C 180,E1 12183.754,E2 12183.754} C_VEL
LIN {X 0,Y 239.137,Z 990.928,A -85,B 0,C 180,E1 12178.192,E2 12178.192} C_VEL
LIN {X 0,Y 235.736,Z 997.713,A -85,B 0,C 180,E1 12173.23,E2 12173.23} C_VEL
LIN {X 0,Y 233.261,Z 1004.018,A -85,B 0,C 180,E1 12167.202,E2 12167.202} C_VEL
LIN {X 0,Y 232.291,Z 1007.738,A -85,B 0,C 180,E1 12162.293,E2 12162.293} C_VEL
LIN {X 0,Y 231.987,Z 1010.435,A -85,B 0,C 180,E1 12156.931,E2 12156.931} C_VEL
LIN {X 0,Y 232.008,Z 1011.514,A -85,B 0,C 180,E1 12152.223,E2 12152.223} C_VEL
LIN {X 0,Y 232.016,Z 1011.561,A -85,B 0,C 180,E1 12148.272,E2 12148.272} C_VEL
LIN {X 0,Y 231.989,Z 1010.719,A -85,B 0,C 180,E1 12144.064,E2 12144.064} C_VEL
LIN {X 0,Y 232.156,Z 1008.607,A -85,B 0,C 180,E1 12139.078,E2 12139.078} C_VEL
LIN {X 0,Y 232.983,Z 1004.864,A -85,B 0,C 180,E1 12133.805,E2 12133.805} C_VEL
LIN {X 0,Y 234.732,Z 1000.026,A -85,B 0,C 180,E1 12128.776,E2 12128.776} C_VEL
LIN {X 0,Y 238.163,Z 992.722,A -85,B 0,C 180,E1 12123.042,E2 12123.042} C_VEL
LIN {X 0,Y 242.819,Z 984.436,A -85,B 0,C 180,E1 12117.919,E2 12117.919} C_VEL
LIN {X 0,Y 248.993,Z 974.32,A -85,B 0,C 180,E1 12112.968,E2 12112.968} C_VEL
LIN {X 0,Y 256.314,Z 963.042,A -85,B 0,C 180,E1 12108.466,E2 12108.466} C_VEL
LIN {X 0,Y 264.623,Z 950.169,A -85,B 0,C 180,E1 12104.347,E2 12104.347} C_VEL
LIN {X 0,Y 273.85,Z 935.874,A -85,B 0,C 180,E1 12100.595,E2 12100.595} C_VEL
LIN {X 0,Y 283.417,Z 920.293,A -85,B 0,C 180,E1 12097.304,E2 12097.304} C_VEL
LIN {X 0,Y 293.833,Z 902.398,A -85,B 0,C 180,E1 12094.231,E2 12094.231} C_VEL
LIN {X 0,Y 302.97,Z 885.485,A -85,B 0,C 180,E1 12091.872,E2 12091.872} C_VEL
LIN {X 0,Y 312.79,Z 865.538,A -85,B 0,C 180,E1 12089.616,E2 12089.616} C_VEL
LIN {X 0,Y 321.675,Z 845.603,A -85,B 0,C 180,E1 12087.79,E2 12087.79} C_VEL
LIN {X 0,Y 329.635,Z 824.972,A -85,B 0,C 180,E1 12086.285,E2 12086.285} C_VEL
LIN {X 0,Y 337.014,Z 803.072,A -85,B 0,C 180,E1 12085.008,E2 12085.008} C_VEL
LIN {X 0,Y 342.99,Z 781.629,A -85,B 0,C 180,E1 12084.038,E2 12084.038} C_VEL
LIN {X 0,Y 348.486,Z 757.03,A -85,B 0,C 180,E1 12083.207,E2 12083.207} C_VEL
LIN {X 0,Y 352.224,Z 734.056,A -85,B 0,C 180,E1 12082.619,E2 12082.619} C_VEL
LIN {X 0,Y 356.061,Z 692.231,A -85,B 0,C 180,E1 12081.776,E2 12081.776} C_VEL
LIN {X 0,Y 368.286,Z 548.523,A -85,B 0,C 180,E1 12078.992,E2 12078.992} C_VEL
LIN {X 0,Y 364.742,Z 541.708,A -85,B 0,C 180,E1 12076.892,E2 12076.892} C_VEL
LIN {X 0,Y 360.039,Z 533.847,A -85,B 0,C 180,E1 12073.653,E2 12073.653} C_VEL
LIN {X 0,Y 356.912,Z 528.995,A -85,B 0,C 180,E1 12070.981,E2 12070.981} C_VEL
LIN {X 0,Y 354.223,Z 524.616,A -85,B 0,C 180,E1 12067.95,E2 12067.95} C_VEL
LIN {X 0,Y 351.926,Z 520.672,A -85,B 0,C 180,E1 12063.746,E2 12063.746} C_VEL
LIN {X 0,Y 351.678,Z 519.666,A -85,B 0,C 180,E1 12062.77,E2 12062.77} C_VEL
LIN {X 0,Y 351.729,Z 519.697,A -85,B 0,C 180,E1 12056.496,E2 12056.496} C_VEL
LIN {X 0,Y 353.791,Z 524.193,A -85,B 0,C 180,E1 12052.04,E2 12052.04} C_VEL
LIN {X 0,Y 354.729,Z 525.353,A -85,B 0,C 180,E1 12050.836,E2 12050.836} C_VEL
LIN {X 0,Y 357.768,Z 530.294,A -85,B 0,C 180,E1 12047.655,E2 12047.655} C_VEL
LIN {X 0,Y 360.849,Z 535.343,A -85,B 0,C 180,E1 12045.149,E2 12045.149} C_VEL
LIN {X 0,Y 364.991,Z 542.174,A -85,B 0,C 180,E1 12042.38,E2 12042.38} C_VEL
LIN {X 0,Y 368.167,Z 547.927,A -85,B 0,C 180,E1 12040.523,E2 12040.523} C_VEL
LIN {X 0,Y 353.264,Z 719.961,A -85,B 0,C 180,E1 12037.19,E2 12037.19} C_VEL
LIN {X 0,Y 349.705,Z 743.741,A -85,B 0,C 180,E1 12036.575,E2 12036.575} C_VEL
LIN {X 0,Y 345.521,Z 764.444,A -85,B 0,C 180,E1 12035.854,E2 12035.854} C_VEL
LIN {X 0,Y 340.035,Z 785.611,A -85,B 0,C 180,E1 12034.897,E2 12034.897} C_VEL
LIN {X 0,Y 333.82,Z 805.731,A -85,B 0,C 180,E1 12033.76,E2 12033.76} C_VEL
LIN {X 0,Y 326.293,Z 826.283,A -85,B 0,C 180,E1 12032.309,E2 12032.309} C_VEL
LIN {X 0,Y 318.369,Z 845.348,A -85,B 0,C 180,E1 12030.664,E2 12030.664} C_VEL
LIN {X 0,Y 309.41,Z 864.276,A -85,B 0,C 180,E1 12028.649,E2 12028.649} C_VEL
LIN {X 0,Y 299.907,Z 882.598,A -85,B 0,C 180,E1 12026.274,E2 12026.274} C_VEL
LIN {X 0,Y 290.471,Z 899.009,A -85,B 0,C 180,E1 12023.646,E2 12023.646} C_VEL
LIN {X 0,Y 280.826,Z 914.783,A -85,B 0,C 180,E1 12020.58,E2 12020.58} C_VEL
LIN {X 0,Y 271.951,Z 928.389,A -85,B 0,C 180,E1 12017.326,E2 12017.326} C_VEL
LIN {X 0,Y 262.61,Z 942.267,A -85,B 0,C 180,E1 12013.254,E2 12013.254} C_VEL
LIN {X 0,Y 254.866,Z 953.51,A -85,B 0,C 180,E1 12009.163,E2 12009.163} C_VEL
LIN {X 0,Y 247.38,Z 964.482,A -85,B 0,C 180,E1 12004.176,E2 12004.176} C_VEL
LIN {X 0,Y 241.514,Z 973.587,A -85,B 0,C 180,E1 11998.967,E2 11998.967} C_VEL
LIN {X 0,Y 237.214,Z 980.759,A -85,B 0,C 180,E1 11993.601,E2 11993.601} C_VEL
LIN {X 0,Y 234.395,Z 986.434,A -85,B 0,C 180,E1 11988.141,E2 11988.141} C_VEL
LIN {X 0,Y 232.862,Z 990.271,A -85,B 0,C 180,E1 11982.899,E2 11982.899} C_VEL
LIN {X 0,Y 232.213,Z 992.777,A -85,B 0,C 180,E1 11977.918,E2 11977.918} C_VEL
LIN {X 0,Y 232.025,Z 994.079,A -85,B 0,C 180,E1 11972.716,E2 11972.716} C_VEL
LIN {X 0,Y 232.026,Z 994.173,A -85,B 0,C 180,E1 11968.271,E2 11968.271} C_VEL
LIN {X 0,Y 232.12,Z 993.361,A -85,B 0,C 180,E1 11963.818,E2 11963.818} C_VEL
LIN {X 0,Y 232.589,Z 991.238,A -85,B 0,C 180,E1 11958.561,E2 11958.561} C_VEL
LIN {X 0,Y 233.825,Z 987.674,A -85,B 0,C 180,E1 11953.306,E2 11953.306} C_VEL
LIN {X 0,Y 236.261,Z 982.643,A -85,B 0,C 180,E1 11947.876,E2 11947.876} C_VEL
LIN {X 0,Y 240.112,Z 975.804,A -85,B 0,C 180,E1 11942.472,E2 11942.472} C_VEL
LIN {X 0,Y 245.542,Z 967.347,A -85,B 0,C 180,E1 11937.212,E2 11937.212} C_VEL
LIN {X 0,Y 252.22,Z 957.434,A -85,B 0,C 180,E1 11932.379,E2 11932.379} C_VEL
LIN {X 0,Y 260.335,Z 945.627,A -85,B 0,C 180,E1 11927.775,E2 11927.775} C_VEL
LIN {X 0,Y 268.906,Z 933.116,A -85,B 0,C 180,E1 11923.841,E2 11923.841} C_VEL
LIN {X 0,Y 277.99,Z 919.269,A -85,B 0,C 180,E1 11920.321,E2 11920.321} C_VEL
LIN {X 0,Y 287.415,Z 904.317,A -85,B 0,C 180,E1 11917.197,E2 11917.197} C_VEL
LIN {X 0,Y 296.95,Z 887.951,A -85,B 0,C 180,E1 11914.427,E2 11914.427} C_VEL
LIN {X 0,Y 306.464,Z 870.463,A -85,B 0,C 180,E1 11911.986,E2 11911.986} C_VEL
LIN {X 0,Y 315.415,Z 852.003,A -85,B 0,C 180,E1 11909.9,E2 11909.9} C_VEL
LIN {X 0,Y 324.047,Z 832.296,A -85,B 0,C 180,E1 11908.07,E2 11908.07} C_VEL
LIN {X 0,Y 331.144,Z 813.661,A -85,B 0,C 180,E1 11906.664,E2 11906.664} C_VEL
LIN {X 0,Y 332.877,Z 808.899,A -85,B 0,C 180,E1 11906.342,E2 11906.342} C_VEL
LIN {X 0,Y 334.815,Z 802.2,A -85,B 0,C 180,E1 11905.751,E2 11905.751} C_VEL
LIN {X 0,Y 337.475,Z 785.527,A -85,B 0,C 180,E1 11903.886,E2 11903.886} C_VEL
LIN {X 0,Y 338.946,Z 778.487,A -85,B 0,C 180,E1 11903.397,E2 11903.397} C_VEL
LIN {X 0,Y 344.272,Z 756.465,A -85,B 0,C 180,E1 11902.509,E2 11902.509} C_VEL
LIN {X 0,Y 348.725,Z 732.184,A -85,B 0,C 180,E1 11901.783,E2 11901.783} C_VEL
LIN {X 0,Y 351.61,Z 708.789,A -85,B 0,C 180,E1 11901.266,E2 11901.266} C_VEL
LIN {X 0,Y 365.263,Z 552.97,A -85,B 0,C 180,E1 11898.266,E2 11898.266} C_VEL
LIN {X 0,Y 360.66,Z 544.933,A -85,B 0,C 180,E1 11895.27,E2 11895.27} C_VEL
LIN {X 0,Y 357.936,Z 540.433,A -85,B 0,C 180,E1 11893.16,E2 11893.16} C_VEL
LIN {X 0,Y 355.627,Z 536.569,A -85,B 0,C 180,E1 11891.022,E2 11891.022} C_VEL
LIN {X 0,Y 353.198,Z 532.509,A -85,B 0,C 180,E1 11888.138,E2 11888.138} C_VEL
LIN {X 0,Y 350.968,Z 528.286,A -85,B 0,C 180,E1 11883.594,E2 11883.594} C_VEL
LIN {X 0,Y 350.791,Z 527.635,A -85,B 0,C 180,E1 11882.778,E2 11882.778} C_VEL
LIN {X 0,Y 350.872,Z 527.722,A -85,B 0,C 180,E1 11877.387,E2 11877.387} C_VEL
LIN {X 0,Y 352.509,Z 531.75,A -85,B 0,C 180,E1 11873.322,E2 11873.322} C_VEL
LIN {X 0,Y 353.67,Z 533.253,A -85,B 0,C 180,E1 11871.711,E2 11871.711} C_VEL
LIN {X 0,Y 356.677,Z 538.321,A -85,B 0,C 180,E1 11868.438,E2 11868.438} C_VEL
LIN {X 0,Y 359.685,Z 543.399,A -85,B 0,C 180,E1 11865.923,E2 11865.923} C_VEL
LIN {X 0,Y 363.264,Z 549.411,A -85,B 0,C 180,E1 11863.449,E2 11863.449} C_VEL
LIN {X 0,Y 365.417,Z 553.797,A -85,B 0,C 180,E1 11862.091,E2 11862.091} C_VEL
LIN {X 0,Y 349.82,Z 729.652,A -85,B 0,C 180,E1 11858.698,E2 11858.698} C_VEL
LIN {X 0,Y 346.098,Z 753.744,A -85,B 0,C 180,E1 11858.11,E2 11858.11} C_VEL
LIN {X 0,Y 341.339,Z 775.932,A -85,B 0,C 180,E1 11857.42,E2 11857.42} C_VEL
LIN {X 0,Y 335.246,Z 797.948,A -85,B 0,C 180,E1 11856.492,E2 11856.492} C_VEL
LIN {X 0,Y 328.328,Z 819.122,A -85,B 0,C 180,E1 11855.357,E2 11855.357} C_VEL
LIN {X 0,Y 320.437,Z 839.481,A -85,B 0,C 180,E1 11853.968,E2 11853.968} C_VEL
LIN {X 0,Y 311.694,Z 859.5,A -85,B 0,C 180,E1 11852.282,E2 11852.282} C_VEL
LIN {X 0,Y 302.561,Z 878.001,A -85,B 0,C 180,E1 11850.346,E2 11850.346} C_VEL
LIN {X 0,Y 291.848,Z 897.721,A -85,B 0,C 180,E1 11847.792,E2 11847.792} C_VEL
LIN {X 0,Y 282.069,Z 914.291,A -85,B 0,C 180,E1 11845.137,E2 11845.137} C_VEL
LIN {X 0,Y 271.8,Z 930.497,A -85,B 0,C 180,E1 11841.92,E2 11841.92} C_VEL
LIN {X 0,Y 262.19,Z 945.102,A -85,B 0,C 180,E1 11838.363,E2 11838.363} C_VEL
LIN {X 0,Y 253.119,Z 958.282,A -85,B 0,C 180,E1 11834.355,E2 11834.355} C_VEL
LIN {X 0,Y 244.908,Z 970.355,A -85,B 0,C 180,E1 11829.859,E2 11829.859} C_VEL
LIN {X 0,Y 237.783,Z 980.956,A -85,B 0,C 180,E1 11824.877,E2 11824.877} C_VEL
LIN {X 0,Y 231.807,Z 990.616,A -85,B 0,C 180,E1 11819.167,E2 11819.167} C_VEL
LIN {X 0,Y 228.125,Z 997.403,A -85,B 0,C 180,E1 11814.053,E2 11814.053} C_VEL
LIN {X 0,Y 225.504,Z 1003.495,A -85,B 0,C 180,E1 11808.08,E2 11808.08} C_VEL
LIN {X 0,Y 224.363,Z 1007.344,A -85,B 0,C 180,E1 11802.874,E2 11802.874} C_VEL
LIN {X 0,Y 223.988,Z 1010.06,A -85,B 0,C 180,E1 11797.438,E2 11797.438} C_VEL
LIN {X 0,Y 224.003,Z 1011.19,A -85,B 0,C 180,E1 11792.559,E2 11792.559} C_VEL
LIN {X 0,Y 224.02,Z 1011.285,A -85,B 0,C 180,E1 11788.466,E2 11788.466} C_VEL
LIN {X 0,Y 223.992,Z 1010.489,A -85,B 0,C 180,E1 11784.109,E2 11784.109} C_VEL
LIN {X 0,Y 224.144,Z 1008.542,A -85,B 0,C 180,E1 11779.204,E2 11779.204} C_VEL
LIN {X 0,Y 225.049,Z 1004.771,A -85,B 0,C 180,E1 11773.483,E2 11773.483} C_VEL
LIN {X 0,Y 226.912,Z 999.979,A -85,B 0,C 180,E1 11768.279,E2 11768.279} C_VEL
LIN {X 0,Y 230.764,Z 992.409,A -85,B 0,C 180,E1 11762.103,E2 11762.103} C_VEL
LIN {X 0,Y 235.768,Z 984.121,A -85,B 0,C 180,E1 11756.839,E2 11756.839} C_VEL
LIN {X 0,Y 242.342,Z 974.004,A -85,B 0,C 180,E1 11751.772,E2 11751.772} C_VEL
LIN {X 0,Y 250.09,Z 962.726,A -85,B 0,C 180,E1 11747.19,E2 11747.19} C_VEL
LIN {X 0,Y 258.691,Z 950.06,A -85,B 0,C 180,E1 11743.08,E2 11743.08} C_VEL
LIN {X 0,Y 268.488,Z 935.558,A -85,B 0,C 180,E1 11739.24,E2 11739.24} C_VEL
LIN {X 0,Y 278.427,Z 919.998,A -85,B 0,C 180,E1 11735.943,E2 11735.943} C_VEL
LIN {X 0,Y 289.275,Z 902.034,A -85,B 0,C 180,E1 11732.864,E2 11732.864} C_VEL
LIN {X 0,Y 298.785,Z 885,A -85,B 0,C 180,E1 11730.504,E2 11730.504} C_VEL
LIN {X 0,Y 308.813,Z 865.226,A -85,B 0,C 180,E1 11728.29,E2 11728.29} C_VEL
LIN {X 0,Y 317.798,Z 845.62,A -85,B 0,C 180,E1 11726.514,E2 11726.514} C_VEL
LIN {X 0,Y 326.014,Z 824.924,A -85,B 0,C 180,E1 11725.02,E2 11725.02} C_VEL
LIN {X 0,Y 333.284,Z 804.051,A -85,B 0,C 180,E1 11723.81,E2 11723.81} C_VEL
LIN {X 0,Y 339.52,Z 782.293,A -85,B 0,C 180,E1 11722.832,E2 11722.832} C_VEL
LIN {X 0,Y 345.024,Z 758.657,A -85,B 0,C 180,E1 11722.033,E2 11722.033} C_VEL
LIN {X 0,Y 348.794,Z 736.507,A -85,B 0,C 180,E1 11721.465,E2 11721.465} C_VEL
LIN {X 0,Y 352.058,Z 704.675,A -85,B 0,C 180,E1 11720.81,E2 11720.81} C_VEL
LIN {X 0,Y 365.268,Z 553.418,A -85,B 0,C 180,E1 11717.894,E2 11717.894} C_VEL
LIN {X 0,Y 361.763,Z 547.022,A -85,B 0,C 180,E1 11715.674,E2 11715.674} C_VEL
LIN {X 0,Y 357.948,Z 540.58,A -85,B 0,C 180,E1 11712.83,E2 11712.83} C_VEL
LIN {X 0,Y 355.597,Z 536.695,A -85,B 0,C 180,E1 11710.694,E2 11710.694} C_VEL
LIN {X 0,Y 353.123,Z 532.494,A -85,B 0,C 180,E1 11707.811,E2 11707.811} C_VEL
LIN {X 0,Y 350.889,Z 528.567,A -85,B 0,C 180,E1 11703.594,E2 11703.594} C_VEL
LIN {X 0,Y 350.654,Z 527.591,A -85,B 0,C 180,E1 11702.615,E2 11702.615} C_VEL
LIN {X 0,Y 350.721,Z 527.691,A -85,B 0,C 180,E1 11696.567,E2 11696.567} C_VEL
LIN {X 0,Y 352.817,Z 532.197,A -85,B 0,C 180,E1 11692.018,E2 11692.018} C_VEL
LIN {X 0,Y 353.61,Z 533.321,A -85,B 0,C 180,E1 11690.971,E2 11690.971} C_VEL
LIN {X 0,Y 356.43,Z 538.003,A -85,B 0,C 180,E1 11687.937,E2 11687.937} C_VEL
LIN {X 0,Y 359.331,Z 542.892,A -85,B 0,C 180,E1 11685.497,E2 11685.497} C_VEL
LIN {X 0,Y 363.243,Z 549.55,A -85,B 0,C 180,E1 11682.788,E2 11682.788} C_VEL
LIN {X 0,Y 365.137,Z 553.132,A -85,B 0,C 180,E1 11681.614,E2 11681.614} C_VEL
LIN {X 0,Y 350.24,Z 720.288,A -85,B 0,C 180,E1 11678.396,E2 11678.396} C_VEL
LIN {X 0,Y 346.625,Z 743.925,A -85,B 0,C 180,E1 11677.793,E2 11677.793} C_VEL
LIN {X 0,Y 342.366,Z 764.54,A -85,B 0,C 180,E1 11677.087,E2 11677.087} C_VEL
LIN {X 0,Y 336.702,Z 785.921,A -85,B 0,C 180,E1 11676.136,E2 11676.136} C_VEL
LIN {X 0,Y 330.334,Z 806.04,A -85,B 0,C 180,E1 11675.015,E2 11675.015} C_VEL
LIN {X 0,Y 322.613,Z 826.592,A -85,B 0,C 180,E1 11673.582,E2 11673.582} C_VEL
LIN {X 0,Y 314.044,Z 846.644,A -85,B 0,C 180,E1 11671.861,E2 11671.861} C_VEL
LIN {X 0,Y 304.706,Z 865.649,A -85,B 0,C 180,E1 11669.83,E2 11669.83} C_VEL
LIN {X 0,Y 294.951,Z 883.744,A -85,B 0,C 180,E1 11667.468,E2 11667.468} C_VEL
LIN {X 0,Y 285.381,Z 899.819,A -85,B 0,C 180,E1 11664.883,E2 11664.883} C_VEL
LIN {X 0,Y 274.54,Z 916.758,A -85,B 0,C 180,E1 11661.528,E2 11661.528} C_VEL
LIN {X 0,Y 265.119,Z 930.628,A -85,B 0,C 180,E1 11658.123,E2 11658.123} C_VEL
